REGION Network 2: DESCRIPTION
   // The block is used as a calling interface for the function blocks  
   // *   _Shiftmodel
   // *   _ProdDataCycleTimer
   // *   _ProdDataCounter
   // *   _ProdDataLimitValues
   // *   _ProdDataShiftCounter
   // or
   // *   _ProdDataShiftCounterOee, ShiftProductionTimes
   // 
   // **Calling interface**  
   // The block must be called once only in the cyclic program.  
   // 
   // The block is used as a calling interface for the function blocks  
   // *   _Shiftmodel
   // *   _ProdDataCycleTimer
   // *   _ProdDataCounter
   // *   _ProdDataLimitValues
   // *   _ProdDataShiftCounter
   // or
   // *   _ProdDataShiftCounterOee, ShiftProductionTimes
   // 
   // #### Additional information
   // 
   // #### Update info
   // 
   // #### Further documentations
   // 
   // ![Icon](_Icon/reference.PNG) 
   // 
   // See:  
   // ..\Library Types\LSicar_Shiftmodel.pdf  
   // ..\Library Types\LSicar_ProdDataCycleTimer.pdf  
   // ..\Library Types\LSicar_ProdDataCounter.pdf  
   // ..\Library Types\LSicar_ProdDataLimitValues.pdf  
   // ..\Library Types\LSicar_ProdDataShiftCounter.pdf  
   // ..\Library Types\LSicar_ProdDataShiftCounterOee.pdf  
   // ..\Library Types\LSicar_ShiftProductionTimes.pdf
END_REGION

REGION Network 3
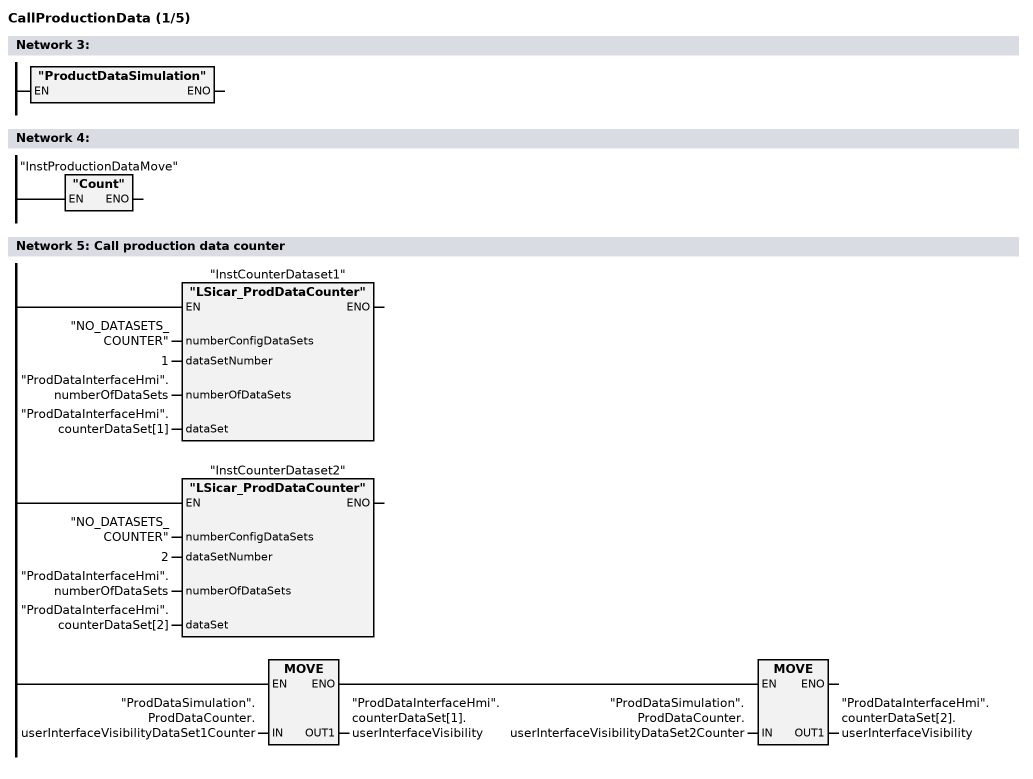
   RUNG wire#powerrail
      "ProductDataSimulation"()
   END_RUNG
   // the same network as SCL:
   "ProductDataSimulation"();
END_REGION

REGION Network 4
   RUNG wire#powerrail
      "InstProductionDataMove"()
   END_RUNG
   // the same network as SCL:
   "InstProductionDataMove"();   // "Count"
END_REGION

REGION Network 5: Call production data counter
   RUNG wire#powerrail
      "InstCounterDataset1"(numberConfigDataSets := "NO_DATASETS_COUNTER", dataSetNumber := 1, numberOfDataSets := "ProdDataInterfaceHmi".numberOfDataSets, dataSet := "ProdDataInterfaceHmi".counterDataSet[1])
   END_RUNG
   RUNG wire#powerrail
      "InstCounterDataset2"(numberConfigDataSets := "NO_DATASETS_COUNTER", dataSetNumber := 2, numberOfDataSets := "ProdDataInterfaceHmi".numberOfDataSets, dataSet := "ProdDataInterfaceHmi".counterDataSet[2])
   END_RUNG
   RUNG wire#powerrail
      Move(in := "ProdDataSimulation".ProdDataCounter.userInterfaceVisibilityDataSet1Counter, out1 => "ProdDataInterfaceHmi".counterDataSet[1].userInterfaceVisibility)
      Move(in := "ProdDataSimulation".ProdDataCounter.userInterfaceVisibilityDataSet2Counter, out1 => "ProdDataInterfaceHmi".counterDataSet[2].userInterfaceVisibility)
   END_RUNG
   // the same network as SCL:
   "InstCounterDataset1"(numberConfigDataSets := "NO_DATASETS_COUNTER",   // "LSicar_ProdDataCounter"
                         dataSetNumber := 1,
                         numberOfDataSets := "ProdDataInterfaceHmi".numberOfDataSets,
                         dataSet := "ProdDataInterfaceHmi".counterDataSet[1]);
   "InstCounterDataset2"(numberConfigDataSets := "NO_DATASETS_COUNTER",   // "LSicar_ProdDataCounter"
                         dataSetNumber := 2,
                         numberOfDataSets := "ProdDataInterfaceHmi".numberOfDataSets,
                         dataSet := "ProdDataInterfaceHmi".counterDataSet[2]);
   "ProdDataInterfaceHmi".counterDataSet[1].userInterfaceVisibility := "ProdDataSimulation".ProdDataCounter.userInterfaceVisibilityDataSet1Counter;
   "ProdDataInterfaceHmi".counterDataSet[2].userInterfaceVisibility := "ProdDataSimulation".ProdDataCounter.userInterfaceVisibilityDataSet2Counter;
END_REGION

REGION Network 6: Call production data cycle timer
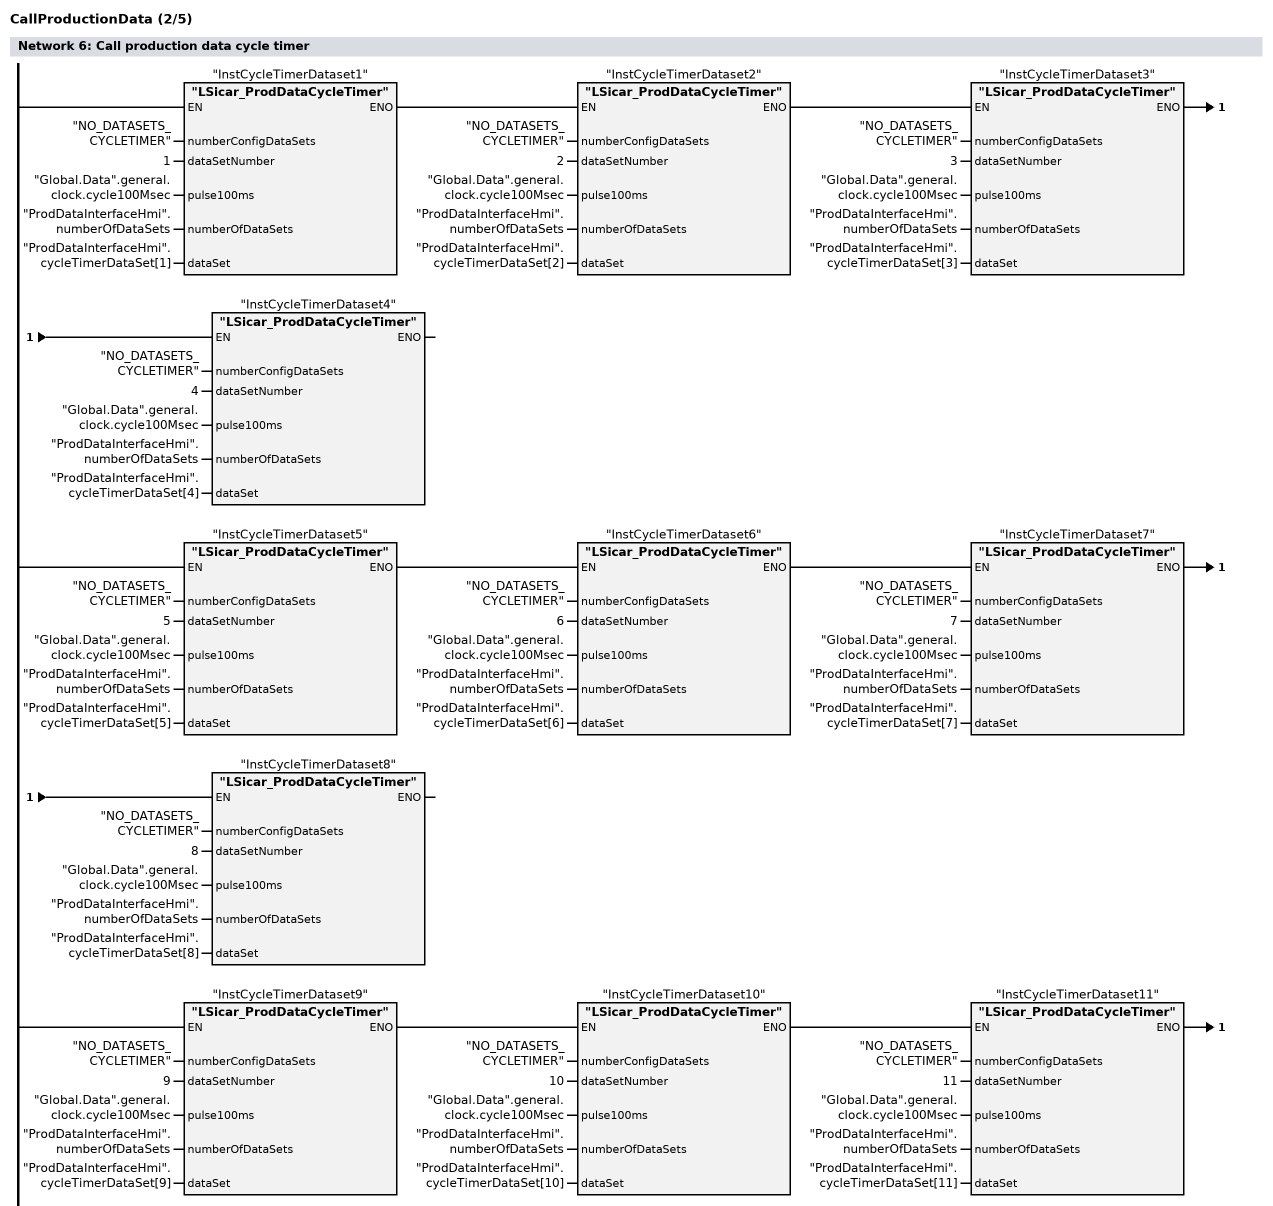
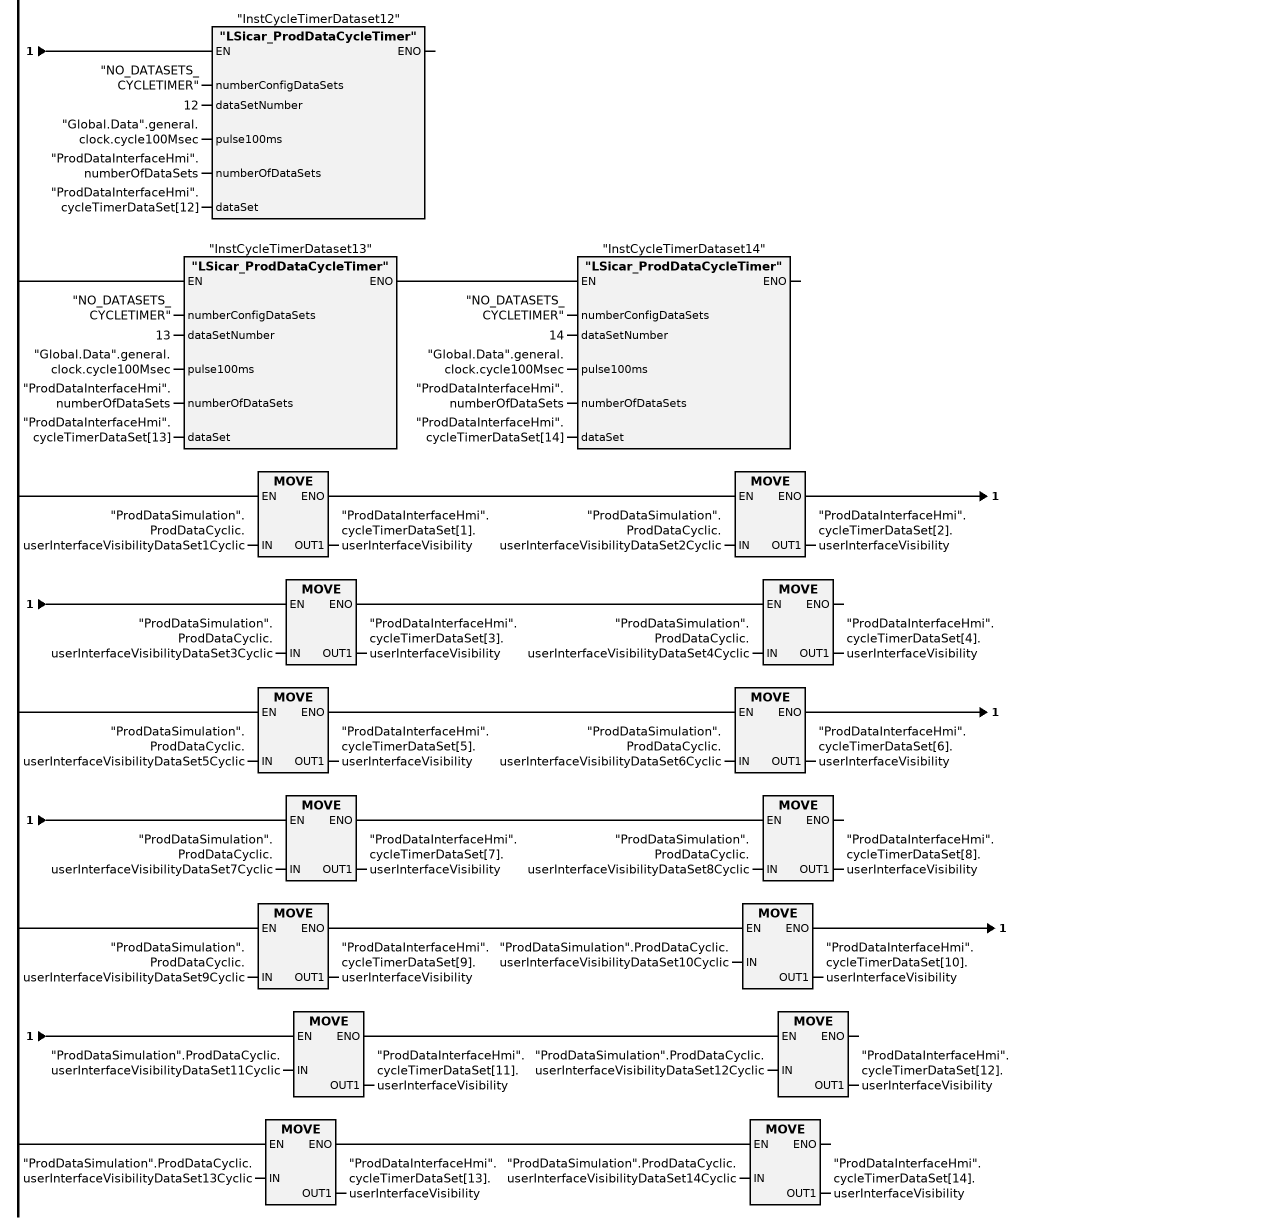
   RUNG wire#powerrail
      "InstCycleTimerDataset1"(numberConfigDataSets := "NO_DATASETS_CYCLETIMER", dataSetNumber := 1, pulse100ms := "Global.Data".general.clock.cycle100Msec, numberOfDataSets := "ProdDataInterfaceHmi".numberOfDataSets, dataSet := "ProdDataInterfaceHmi".cycleTimerDataSet[1])
      "InstCycleTimerDataset2"(numberConfigDataSets := "NO_DATASETS_CYCLETIMER", dataSetNumber := 2, pulse100ms := "Global.Data".general.clock.cycle100Msec, numberOfDataSets := "ProdDataInterfaceHmi".numberOfDataSets, dataSet := "ProdDataInterfaceHmi".cycleTimerDataSet[2])
      "InstCycleTimerDataset3"(numberConfigDataSets := "NO_DATASETS_CYCLETIMER", dataSetNumber := 3, pulse100ms := "Global.Data".general.clock.cycle100Msec, numberOfDataSets := "ProdDataInterfaceHmi".numberOfDataSets, dataSet := "ProdDataInterfaceHmi".cycleTimerDataSet[3])
      "InstCycleTimerDataset4"(numberConfigDataSets := "NO_DATASETS_CYCLETIMER", dataSetNumber := 4, pulse100ms := "Global.Data".general.clock.cycle100Msec, numberOfDataSets := "ProdDataInterfaceHmi".numberOfDataSets, dataSet := "ProdDataInterfaceHmi".cycleTimerDataSet[4])
   END_RUNG
   RUNG wire#powerrail
      "InstCycleTimerDataset5"(numberConfigDataSets := "NO_DATASETS_CYCLETIMER", dataSetNumber := 5, pulse100ms := "Global.Data".general.clock.cycle100Msec, numberOfDataSets := "ProdDataInterfaceHmi".numberOfDataSets, dataSet := "ProdDataInterfaceHmi".cycleTimerDataSet[5])
      "InstCycleTimerDataset6"(numberConfigDataSets := "NO_DATASETS_CYCLETIMER", dataSetNumber := 6, pulse100ms := "Global.Data".general.clock.cycle100Msec, numberOfDataSets := "ProdDataInterfaceHmi".numberOfDataSets, dataSet := "ProdDataInterfaceHmi".cycleTimerDataSet[6])
      "InstCycleTimerDataset7"(numberConfigDataSets := "NO_DATASETS_CYCLETIMER", dataSetNumber := 7, pulse100ms := "Global.Data".general.clock.cycle100Msec, numberOfDataSets := "ProdDataInterfaceHmi".numberOfDataSets, dataSet := "ProdDataInterfaceHmi".cycleTimerDataSet[7])
      "InstCycleTimerDataset8"(numberConfigDataSets := "NO_DATASETS_CYCLETIMER", dataSetNumber := 8, pulse100ms := "Global.Data".general.clock.cycle100Msec, numberOfDataSets := "ProdDataInterfaceHmi".numberOfDataSets, dataSet := "ProdDataInterfaceHmi".cycleTimerDataSet[8])
   END_RUNG
   RUNG wire#powerrail
      "InstCycleTimerDataset9"(numberConfigDataSets := "NO_DATASETS_CYCLETIMER", dataSetNumber := 9, pulse100ms := "Global.Data".general.clock.cycle100Msec, numberOfDataSets := "ProdDataInterfaceHmi".numberOfDataSets, dataSet := "ProdDataInterfaceHmi".cycleTimerDataSet[9])
      "InstCycleTimerDataset10"(numberConfigDataSets := "NO_DATASETS_CYCLETIMER", dataSetNumber := 10, pulse100ms := "Global.Data".general.clock.cycle100Msec, numberOfDataSets := "ProdDataInterfaceHmi".numberOfDataSets, dataSet := "ProdDataInterfaceHmi".cycleTimerDataSet[10])
      "InstCycleTimerDataset11"(numberConfigDataSets := "NO_DATASETS_CYCLETIMER", dataSetNumber := 11, pulse100ms := "Global.Data".general.clock.cycle100Msec, numberOfDataSets := "ProdDataInterfaceHmi".numberOfDataSets, dataSet := "ProdDataInterfaceHmi".cycleTimerDataSet[11])
      "InstCycleTimerDataset12"(numberConfigDataSets := "NO_DATASETS_CYCLETIMER", dataSetNumber := 12, pulse100ms := "Global.Data".general.clock.cycle100Msec, numberOfDataSets := "ProdDataInterfaceHmi".numberOfDataSets, dataSet := "ProdDataInterfaceHmi".cycleTimerDataSet[12])
   END_RUNG
   RUNG wire#powerrail
      "InstCycleTimerDataset13"(numberConfigDataSets := "NO_DATASETS_CYCLETIMER", dataSetNumber := 13, pulse100ms := "Global.Data".general.clock.cycle100Msec, numberOfDataSets := "ProdDataInterfaceHmi".numberOfDataSets, dataSet := "ProdDataInterfaceHmi".cycleTimerDataSet[13])
      "InstCycleTimerDataset14"(numberConfigDataSets := "NO_DATASETS_CYCLETIMER", dataSetNumber := 14, pulse100ms := "Global.Data".general.clock.cycle100Msec, numberOfDataSets := "ProdDataInterfaceHmi".numberOfDataSets, dataSet := "ProdDataInterfaceHmi".cycleTimerDataSet[14])
   END_RUNG
   RUNG wire#powerrail
      Move(in := "ProdDataSimulation".ProdDataCyclic.userInterfaceVisibilityDataSet1Cyclic, out1 => "ProdDataInterfaceHmi".cycleTimerDataSet[1].userInterfaceVisibility)
      Move(in := "ProdDataSimulation".ProdDataCyclic.userInterfaceVisibilityDataSet2Cyclic, out1 => "ProdDataInterfaceHmi".cycleTimerDataSet[2].userInterfaceVisibility)
      Move(in := "ProdDataSimulation".ProdDataCyclic.userInterfaceVisibilityDataSet3Cyclic, out1 => "ProdDataInterfaceHmi".cycleTimerDataSet[3].userInterfaceVisibility)
      Move(in := "ProdDataSimulation".ProdDataCyclic.userInterfaceVisibilityDataSet4Cyclic, out1 => "ProdDataInterfaceHmi".cycleTimerDataSet[4].userInterfaceVisibility)
   END_RUNG
   RUNG wire#powerrail
      Move(in := "ProdDataSimulation".ProdDataCyclic.userInterfaceVisibilityDataSet5Cyclic, out1 => "ProdDataInterfaceHmi".cycleTimerDataSet[5].userInterfaceVisibility)
      Move(in := "ProdDataSimulation".ProdDataCyclic.userInterfaceVisibilityDataSet6Cyclic, out1 => "ProdDataInterfaceHmi".cycleTimerDataSet[6].userInterfaceVisibility)
      Move(in := "ProdDataSimulation".ProdDataCyclic.userInterfaceVisibilityDataSet7Cyclic, out1 => "ProdDataInterfaceHmi".cycleTimerDataSet[7].userInterfaceVisibility)
      Move(in := "ProdDataSimulation".ProdDataCyclic.userInterfaceVisibilityDataSet8Cyclic, out1 => "ProdDataInterfaceHmi".cycleTimerDataSet[8].userInterfaceVisibility)
   END_RUNG
   RUNG wire#powerrail
      Move(in := "ProdDataSimulation".ProdDataCyclic.userInterfaceVisibilityDataSet9Cyclic, out1 => "ProdDataInterfaceHmi".cycleTimerDataSet[9].userInterfaceVisibility)
      Move(in := "ProdDataSimulation".ProdDataCyclic.userInterfaceVisibilityDataSet10Cyclic, out1 => "ProdDataInterfaceHmi".cycleTimerDataSet[10].userInterfaceVisibility)
      Move(in := "ProdDataSimulation".ProdDataCyclic.userInterfaceVisibilityDataSet11Cyclic, out1 => "ProdDataInterfaceHmi".cycleTimerDataSet[11].userInterfaceVisibility)
      Move(in := "ProdDataSimulation".ProdDataCyclic.userInterfaceVisibilityDataSet12Cyclic, out1 => "ProdDataInterfaceHmi".cycleTimerDataSet[12].userInterfaceVisibility)
   END_RUNG
   RUNG wire#powerrail
      Move(in := "ProdDataSimulation".ProdDataCyclic.userInterfaceVisibilityDataSet13Cyclic, out1 => "ProdDataInterfaceHmi".cycleTimerDataSet[13].userInterfaceVisibility)
      Move(in := "ProdDataSimulation".ProdDataCyclic.userInterfaceVisibilityDataSet14Cyclic, out1 => "ProdDataInterfaceHmi".cycleTimerDataSet[14].userInterfaceVisibility)
   END_RUNG
   // the same network as SCL:
   "InstCycleTimerDataset1"(numberConfigDataSets := "NO_DATASETS_CYCLETIMER",   // "LSicar_ProdDataCycleTimer"
                           dataSetNumber := 1,
                           pulse100ms := "Global.Data".general.clock.cycle100Msec,
                           numberOfDataSets := "ProdDataInterfaceHmi".numberOfDataSets,
                           dataSet := "ProdDataInterfaceHmi".cycleTimerDataSet[1],
                           ENO => #_w1);
   "InstCycleTimerDataset2"(EN := #_w1,   // "LSicar_ProdDataCycleTimer"
                           numberConfigDataSets := "NO_DATASETS_CYCLETIMER",
                           dataSetNumber := 2,
                           pulse100ms := "Global.Data".general.clock.cycle100Msec,
                           numberOfDataSets := "ProdDataInterfaceHmi".numberOfDataSets,
                           dataSet := "ProdDataInterfaceHmi".cycleTimerDataSet[2],
                           ENO => #_w2);
   "InstCycleTimerDataset3"(EN := #_w2,   // "LSicar_ProdDataCycleTimer"
                           numberConfigDataSets := "NO_DATASETS_CYCLETIMER",
                           dataSetNumber := 3,
                           pulse100ms := "Global.Data".general.clock.cycle100Msec,
                           numberOfDataSets := "ProdDataInterfaceHmi".numberOfDataSets,
                           dataSet := "ProdDataInterfaceHmi".cycleTimerDataSet[3],
                           ENO => #_w3);
   IF #_w3 THEN
       "InstCycleTimerDataset4"(numberConfigDataSets := "NO_DATASETS_CYCLETIMER",   // "LSicar_ProdDataCycleTimer"
                               dataSetNumber := 4,
                               pulse100ms := "Global.Data".general.clock.cycle100Msec,
                               numberOfDataSets := "ProdDataInterfaceHmi".numberOfDataSets,
                               dataSet := "ProdDataInterfaceHmi".cycleTimerDataSet[4]);
   END_IF;
   "InstCycleTimerDataset5"(numberConfigDataSets := "NO_DATASETS_CYCLETIMER",   // "LSicar_ProdDataCycleTimer"
                           dataSetNumber := 5,
                           pulse100ms := "Global.Data".general.clock.cycle100Msec,
                           numberOfDataSets := "ProdDataInterfaceHmi".numberOfDataSets,
                           dataSet := "ProdDataInterfaceHmi".cycleTimerDataSet[5],
                           ENO => #_w4);
   "InstCycleTimerDataset6"(EN := #_w4,   // "LSicar_ProdDataCycleTimer"
                           numberConfigDataSets := "NO_DATASETS_CYCLETIMER",
                           dataSetNumber := 6,
                           pulse100ms := "Global.Data".general.clock.cycle100Msec,
                           numberOfDataSets := "ProdDataInterfaceHmi".numberOfDataSets,
                           dataSet := "ProdDataInterfaceHmi".cycleTimerDataSet[6],
                           ENO => #_w5);
   "InstCycleTimerDataset7"(EN := #_w5,   // "LSicar_ProdDataCycleTimer"
                           numberConfigDataSets := "NO_DATASETS_CYCLETIMER",
                           dataSetNumber := 7,
                           pulse100ms := "Global.Data".general.clock.cycle100Msec,
                           numberOfDataSets := "ProdDataInterfaceHmi".numberOfDataSets,
                           dataSet := "ProdDataInterfaceHmi".cycleTimerDataSet[7],
                           ENO => #_w6);
   IF #_w6 THEN
       "InstCycleTimerDataset8"(numberConfigDataSets := "NO_DATASETS_CYCLETIMER",   // "LSicar_ProdDataCycleTimer"
                               dataSetNumber := 8,
                               pulse100ms := "Global.Data".general.clock.cycle100Msec,
                               numberOfDataSets := "ProdDataInterfaceHmi".numberOfDataSets,
                               dataSet := "ProdDataInterfaceHmi".cycleTimerDataSet[8]);
   END_IF;
   "InstCycleTimerDataset9"(numberConfigDataSets := "NO_DATASETS_CYCLETIMER",   // "LSicar_ProdDataCycleTimer"
                           dataSetNumber := 9,
                           pulse100ms := "Global.Data".general.clock.cycle100Msec,
                           numberOfDataSets := "ProdDataInterfaceHmi".numberOfDataSets,
                           dataSet := "ProdDataInterfaceHmi".cycleTimerDataSet[9],
                           ENO => #_w7);
   "InstCycleTimerDataset10"(EN := #_w7,   // "LSicar_ProdDataCycleTimer"
                           numberConfigDataSets := "NO_DATASETS_CYCLETIMER",
                           dataSetNumber := 10,
                           pulse100ms := "Global.Data".general.clock.cycle100Msec,
                           numberOfDataSets := "ProdDataInterfaceHmi".numberOfDataSets,
                           dataSet := "ProdDataInterfaceHmi".cycleTimerDataSet[10],
                           ENO => #_w8);
   "InstCycleTimerDataset11"(EN := #_w8,   // "LSicar_ProdDataCycleTimer"
                           numberConfigDataSets := "NO_DATASETS_CYCLETIMER",
                           dataSetNumber := 11,
                           pulse100ms := "Global.Data".general.clock.cycle100Msec,
                           numberOfDataSets := "ProdDataInterfaceHmi".numberOfDataSets,
                           dataSet := "ProdDataInterfaceHmi".cycleTimerDataSet[11],
                           ENO => #_w9);
   IF #_w9 THEN
       "InstCycleTimerDataset12"(numberConfigDataSets := "NO_DATASETS_CYCLETIMER",   // "LSicar_ProdDataCycleTimer"
                               dataSetNumber := 12,
                               pulse100ms := "Global.Data".general.clock.cycle100Msec,
                               numberOfDataSets := "ProdDataInterfaceHmi".numberOfDataSets,
                               dataSet := "ProdDataInterfaceHmi".cycleTimerDataSet[12]);
   END_IF;
   "InstCycleTimerDataset13"(numberConfigDataSets := "NO_DATASETS_CYCLETIMER",   // "LSicar_ProdDataCycleTimer"
                           dataSetNumber := 13,
                           pulse100ms := "Global.Data".general.clock.cycle100Msec,
                           numberOfDataSets := "ProdDataInterfaceHmi".numberOfDataSets,
                           dataSet := "ProdDataInterfaceHmi".cycleTimerDataSet[13],
                           ENO => #_w10);
   IF #_w10 THEN
       "InstCycleTimerDataset14"(numberConfigDataSets := "NO_DATASETS_CYCLETIMER",   // "LSicar_ProdDataCycleTimer"
                               dataSetNumber := 14,
                               pulse100ms := "Global.Data".general.clock.cycle100Msec,
                               numberOfDataSets := "ProdDataInterfaceHmi".numberOfDataSets,
                               dataSet := "ProdDataInterfaceHmi".cycleTimerDataSet[14]);
   END_IF;
   "ProdDataInterfaceHmi".cycleTimerDataSet[1].userInterfaceVisibility := "ProdDataSimulation".ProdDataCyclic.userInterfaceVisibilityDataSet1Cyclic;
   "ProdDataInterfaceHmi".cycleTimerDataSet[2].userInterfaceVisibility := "ProdDataSimulation".ProdDataCyclic.userInterfaceVisibilityDataSet2Cyclic;
   "ProdDataInterfaceHmi".cycleTimerDataSet[3].userInterfaceVisibility := "ProdDataSimulation".ProdDataCyclic.userInterfaceVisibilityDataSet3Cyclic;
   "ProdDataInterfaceHmi".cycleTimerDataSet[4].userInterfaceVisibility := "ProdDataSimulation".ProdDataCyclic.userInterfaceVisibilityDataSet4Cyclic;
   "ProdDataInterfaceHmi".cycleTimerDataSet[5].userInterfaceVisibility := "ProdDataSimulation".ProdDataCyclic.userInterfaceVisibilityDataSet5Cyclic;
   "ProdDataInterfaceHmi".cycleTimerDataSet[6].userInterfaceVisibility := "ProdDataSimulation".ProdDataCyclic.userInterfaceVisibilityDataSet6Cyclic;
   "ProdDataInterfaceHmi".cycleTimerDataSet[7].userInterfaceVisibility := "ProdDataSimulation".ProdDataCyclic.userInterfaceVisibilityDataSet7Cyclic;
   "ProdDataInterfaceHmi".cycleTimerDataSet[8].userInterfaceVisibility := "ProdDataSimulation".ProdDataCyclic.userInterfaceVisibilityDataSet8Cyclic;
   "ProdDataInterfaceHmi".cycleTimerDataSet[9].userInterfaceVisibility := "ProdDataSimulation".ProdDataCyclic.userInterfaceVisibilityDataSet9Cyclic;
   "ProdDataInterfaceHmi".cycleTimerDataSet[10].userInterfaceVisibility := "ProdDataSimulation".ProdDataCyclic.userInterfaceVisibilityDataSet10Cyclic;
   "ProdDataInterfaceHmi".cycleTimerDataSet[11].userInterfaceVisibility := "ProdDataSimulation".ProdDataCyclic.userInterfaceVisibilityDataSet11Cyclic;
   "ProdDataInterfaceHmi".cycleTimerDataSet[12].userInterfaceVisibility := "ProdDataSimulation".ProdDataCyclic.userInterfaceVisibilityDataSet12Cyclic;
   "ProdDataInterfaceHmi".cycleTimerDataSet[13].userInterfaceVisibility := "ProdDataSimulation".ProdDataCyclic.userInterfaceVisibilityDataSet13Cyclic;
   "ProdDataInterfaceHmi".cycleTimerDataSet[14].userInterfaceVisibility := "ProdDataSimulation".ProdDataCyclic.userInterfaceVisibilityDataSet14Cyclic;
END_REGION

REGION Network 7: Call production data limit values
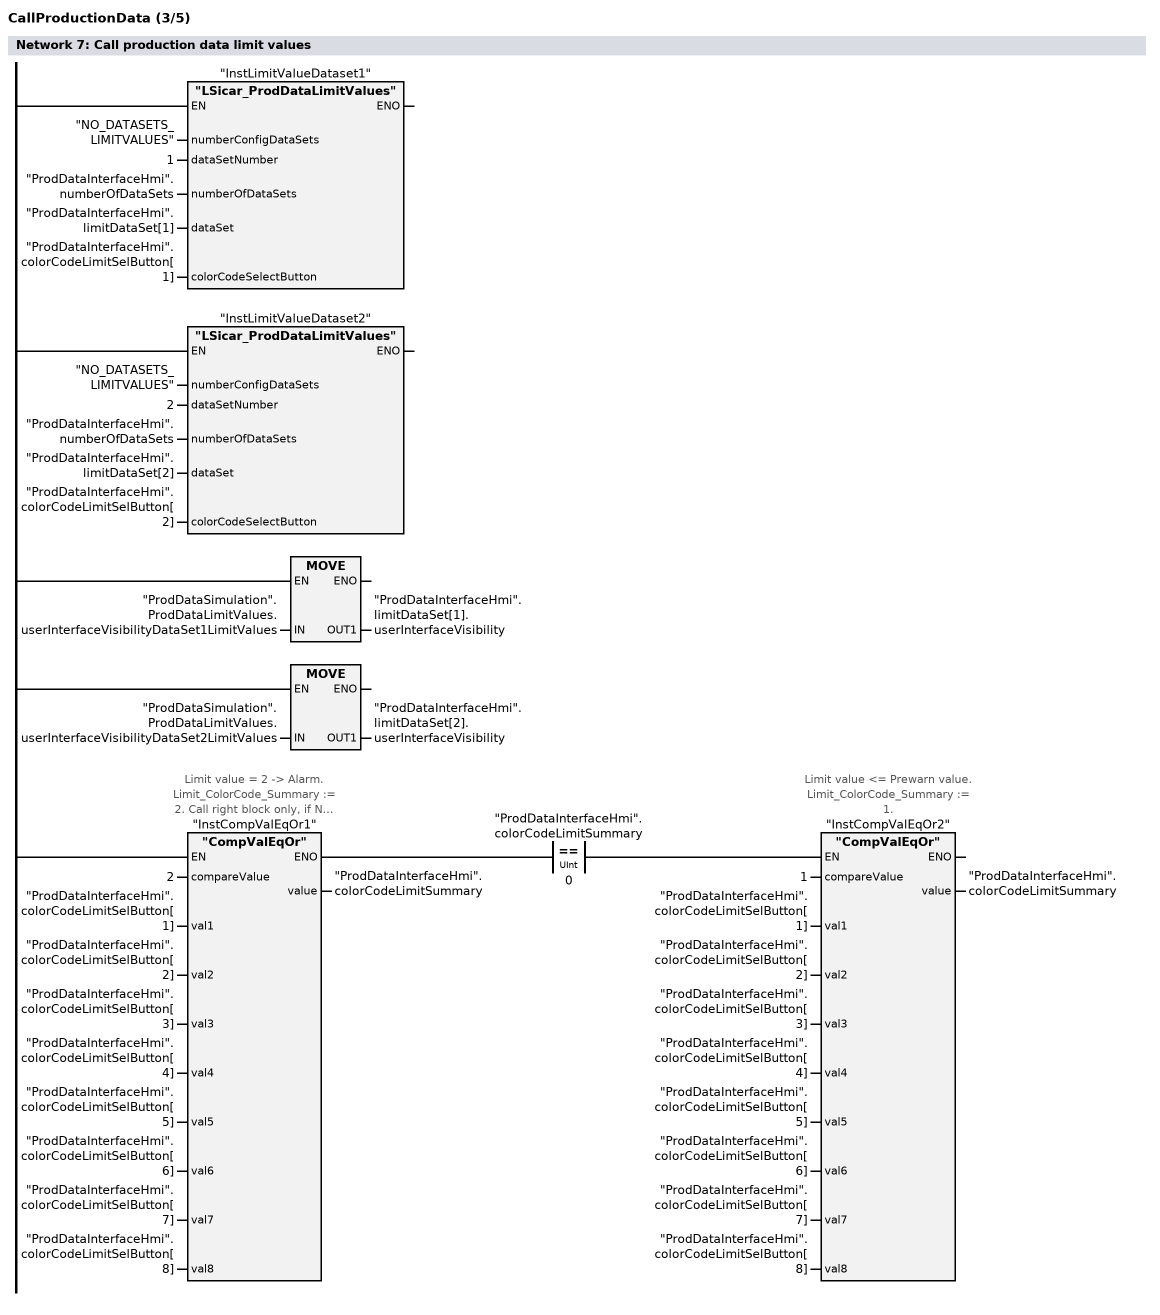
   RUNG wire#powerrail
      "InstLimitValueDataset1"(numberConfigDataSets := "NO_DATASETS_LIMITVALUES", dataSetNumber := 1, numberOfDataSets := "ProdDataInterfaceHmi".numberOfDataSets, dataSet := "ProdDataInterfaceHmi".limitDataSet[1], colorCodeSelectButton := "ProdDataInterfaceHmi".colorCodeLimitSelButton[1])
   END_RUNG
   RUNG wire#powerrail
      "InstLimitValueDataset2"(numberConfigDataSets := "NO_DATASETS_LIMITVALUES", dataSetNumber := 2, numberOfDataSets := "ProdDataInterfaceHmi".numberOfDataSets, dataSet := "ProdDataInterfaceHmi".limitDataSet[2], colorCodeSelectButton := "ProdDataInterfaceHmi".colorCodeLimitSelButton[2])
   END_RUNG
   RUNG wire#powerrail
      Move(in := "ProdDataSimulation".ProdDataLimitValues.userInterfaceVisibilityDataSet1LimitValues, out1 => "ProdDataInterfaceHmi".limitDataSet[1].userInterfaceVisibility)
   END_RUNG
   RUNG wire#powerrail
      Move(in := "ProdDataSimulation".ProdDataLimitValues.userInterfaceVisibilityDataSet2LimitValues, out1 => "ProdDataInterfaceHmi".limitDataSet[2].userInterfaceVisibility)
   END_RUNG
   RUNG wire#powerrail
      "InstCompValEqOr1"(compareValue := 2, val1 := "ProdDataInterfaceHmi".colorCodeLimitSelButton[1], val2 := "ProdDataInterfaceHmi".colorCodeLimitSelButton[2], val3 := "ProdDataInterfaceHmi".colorCodeLimitSelButton[3], val4 := "ProdDataInterfaceHmi".colorCodeLimitSelButton[4], val5 := "ProdDataInterfaceHmi".colorCodeLimitSelButton[5], val6 := "ProdDataInterfaceHmi".colorCodeLimitSelButton[6], val7 := "ProdDataInterfaceHmi".colorCodeLimitSelButton[7], val8 := "ProdDataInterfaceHmi".colorCodeLimitSelButton[8], value => "ProdDataInterfaceHmi".colorCodeLimitSummary)   // Limit value = 2 -> Alarm. Limit_ColorCode_Summary := 2. Call right block only, if NO alarm (VALUE = 0) is pending here; alarm is higher prior.
      { S7_Templates := "SrcType := UInt" } EQ_Contact(in1 := "ProdDataInterfaceHmi".colorCodeLimitSummary, in2 := 0)
      "InstCompValEqOr2"(compareValue := 1, val1 := "ProdDataInterfaceHmi".colorCodeLimitSelButton[1], val2 := "ProdDataInterfaceHmi".colorCodeLimitSelButton[2], val3 := "ProdDataInterfaceHmi".colorCodeLimitSelButton[3], val4 := "ProdDataInterfaceHmi".colorCodeLimitSelButton[4], val5 := "ProdDataInterfaceHmi".colorCodeLimitSelButton[5], val6 := "ProdDataInterfaceHmi".colorCodeLimitSelButton[6], val7 := "ProdDataInterfaceHmi".colorCodeLimitSelButton[7], val8 := "ProdDataInterfaceHmi".colorCodeLimitSelButton[8], value => "ProdDataInterfaceHmi".colorCodeLimitSummary)   // Limit value <= Prewarn value. Limit_ColorCode_Summary := 1.
   END_RUNG
   // the same network as SCL:
   "InstLimitValueDataset1"(numberConfigDataSets := "NO_DATASETS_LIMITVALUES",   // "LSicar_ProdDataLimitValues"
                           dataSetNumber := 1,
                           numberOfDataSets := "ProdDataInterfaceHmi".numberOfDataSets,
                           dataSet := "ProdDataInterfaceHmi".limitDataSet[1],
                           colorCodeSelectButton := "ProdDataInterfaceHmi".colorCodeLimitSelButton[1]);
   "InstLimitValueDataset2"(numberConfigDataSets := "NO_DATASETS_LIMITVALUES",   // "LSicar_ProdDataLimitValues"
                           dataSetNumber := 2,
                           numberOfDataSets := "ProdDataInterfaceHmi".numberOfDataSets,
                           dataSet := "ProdDataInterfaceHmi".limitDataSet[2],
                           colorCodeSelectButton := "ProdDataInterfaceHmi".colorCodeLimitSelButton[2]);
   "ProdDataInterfaceHmi".limitDataSet[1].userInterfaceVisibility := "ProdDataSimulation".ProdDataLimitValues.userInterfaceVisibilityDataSet1LimitValues;
   "ProdDataInterfaceHmi".limitDataSet[2].userInterfaceVisibility := "ProdDataSimulation".ProdDataLimitValues.userInterfaceVisibilityDataSet2LimitValues;
   "InstCompValEqOr1"(compareValue := 2,   // "CompValEqOr": Limit value = 2 -> Alarm. Limit_ColorCode_Summary := 2. Call right block only, if NO alarm (VALUE = 0) is pending here; alarm is higher prior.
                      val1 := "ProdDataInterfaceHmi".colorCodeLimitSelButton[1],
                      val2 := "ProdDataInterfaceHmi".colorCodeLimitSelButton[2],
                      val3 := "ProdDataInterfaceHmi".colorCodeLimitSelButton[3],
                      val4 := "ProdDataInterfaceHmi".colorCodeLimitSelButton[4],
                      val5 := "ProdDataInterfaceHmi".colorCodeLimitSelButton[5],
                      val6 := "ProdDataInterfaceHmi".colorCodeLimitSelButton[6],
                      val7 := "ProdDataInterfaceHmi".colorCodeLimitSelButton[7],
                      val8 := "ProdDataInterfaceHmi".colorCodeLimitSelButton[8],
                      value => "ProdDataInterfaceHmi".colorCodeLimitSummary,
                      ENO => #_w1);
   IF #_w1 AND ("ProdDataInterfaceHmi".colorCodeLimitSummary = 0) THEN
       "InstCompValEqOr2"(compareValue := 1,   // "CompValEqOr": Limit value <= Prewarn value. Limit_ColorCode_Summary := 1.
                          val1 := "ProdDataInterfaceHmi".colorCodeLimitSelButton[1],
                          val2 := "ProdDataInterfaceHmi".colorCodeLimitSelButton[2],
                          val3 := "ProdDataInterfaceHmi".colorCodeLimitSelButton[3],
                          val4 := "ProdDataInterfaceHmi".colorCodeLimitSelButton[4],
                          val5 := "ProdDataInterfaceHmi".colorCodeLimitSelButton[5],
                          val6 := "ProdDataInterfaceHmi".colorCodeLimitSelButton[6],
                          val7 := "ProdDataInterfaceHmi".colorCodeLimitSelButton[7],
                          val8 := "ProdDataInterfaceHmi".colorCodeLimitSelButton[8],
                          value => "ProdDataInterfaceHmi".colorCodeLimitSummary);
   END_IF;
END_REGION

REGION Network 8: Call production data shift counter
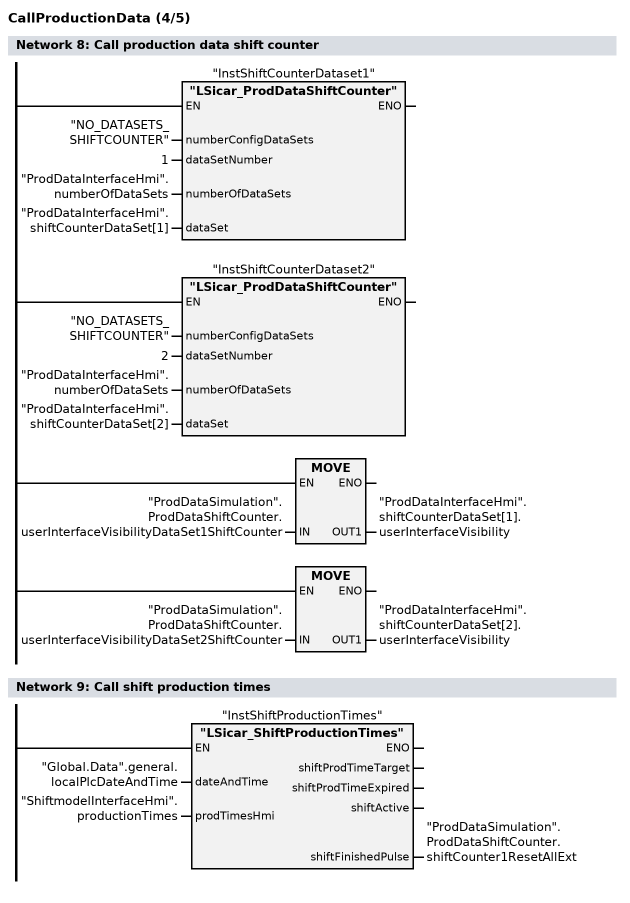
   RUNG wire#powerrail
      "InstShiftCounterDataset1"(numberConfigDataSets := "NO_DATASETS_SHIFTCOUNTER", dataSetNumber := 1, numberOfDataSets := "ProdDataInterfaceHmi".numberOfDataSets, dataSet := "ProdDataInterfaceHmi".shiftCounterDataSet[1])
   END_RUNG
   RUNG wire#powerrail
      "InstShiftCounterDataset2"(numberConfigDataSets := "NO_DATASETS_SHIFTCOUNTER", dataSetNumber := 2, numberOfDataSets := "ProdDataInterfaceHmi".numberOfDataSets, dataSet := "ProdDataInterfaceHmi".shiftCounterDataSet[2])
   END_RUNG
   RUNG wire#powerrail
      Move(in := "ProdDataSimulation".ProdDataShiftCounter.userInterfaceVisibilityDataSet1ShiftCounter, out1 => "ProdDataInterfaceHmi".shiftCounterDataSet[1].userInterfaceVisibility)
   END_RUNG
   RUNG wire#powerrail
      Move(in := "ProdDataSimulation".ProdDataShiftCounter.userInterfaceVisibilityDataSet2ShiftCounter, out1 => "ProdDataInterfaceHmi".shiftCounterDataSet[2].userInterfaceVisibility)
   END_RUNG
   // the same network as SCL:
   "InstShiftCounterDataset1"(numberConfigDataSets := "NO_DATASETS_SHIFTCOUNTER",   // "LSicar_ProdDataShiftCounter"
                           dataSetNumber := 1,
                           numberOfDataSets := "ProdDataInterfaceHmi".numberOfDataSets,
                           dataSet := "ProdDataInterfaceHmi".shiftCounterDataSet[1]);
   "InstShiftCounterDataset2"(numberConfigDataSets := "NO_DATASETS_SHIFTCOUNTER",   // "LSicar_ProdDataShiftCounter"
                           dataSetNumber := 2,
                           numberOfDataSets := "ProdDataInterfaceHmi".numberOfDataSets,
                           dataSet := "ProdDataInterfaceHmi".shiftCounterDataSet[2]);
   "ProdDataInterfaceHmi".shiftCounterDataSet[1].userInterfaceVisibility := "ProdDataSimulation".ProdDataShiftCounter.userInterfaceVisibilityDataSet1ShiftCounter;
   "ProdDataInterfaceHmi".shiftCounterDataSet[2].userInterfaceVisibility := "ProdDataSimulation".ProdDataShiftCounter.userInterfaceVisibilityDataSet2ShiftCounter;
END_REGION

REGION Network 9: Call shift production times
   RUNG wire#powerrail
      "InstShiftProductionTimes"(dateAndTime := "Global.Data".general.localPlcDateAndTime, prodTimesHmi := "ShiftmodelInterfaceHmi".productionTimes, shiftProdTimeTarget =>, shiftProdTimeExpired =>, shiftActive =>, shiftFinishedPulse => "ProdDataSimulation".ProdDataShiftCounter.shiftCounter1ResetAllExt)
   END_RUNG
   // the same network as SCL:
   "InstShiftProductionTimes"(dateAndTime := "Global.Data".general.localPlcDateAndTime,   // "LSicar_ShiftProductionTimes"
                           prodTimesHmi := "ShiftmodelInterfaceHmi".productionTimes,
                           shiftFinishedPulse => "ProdDataSimulation".ProdDataShiftCounter.shiftCounter1ResetAllExt);
END_REGION

REGION Network 10: Call production data shift counter OEE
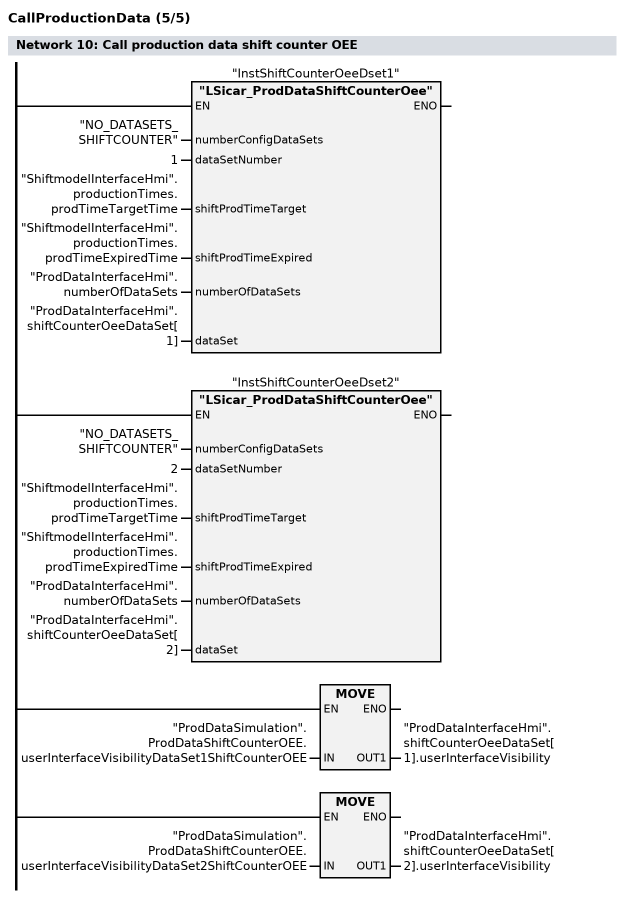
   RUNG wire#powerrail
      "InstShiftCounterOeeDset1"(numberConfigDataSets := "NO_DATASETS_SHIFTCOUNTER", dataSetNumber := 1, shiftProdTimeTarget := "ShiftmodelInterfaceHmi".productionTimes.prodTimeTargetTime, shiftProdTimeExpired := "ShiftmodelInterfaceHmi".productionTimes.prodTimeExpiredTime, numberOfDataSets := "ProdDataInterfaceHmi".numberOfDataSets, dataSet := "ProdDataInterfaceHmi".shiftCounterOeeDataSet[1])
   END_RUNG
   RUNG wire#powerrail
      "InstShiftCounterOeeDset2"(numberConfigDataSets := "NO_DATASETS_SHIFTCOUNTER", dataSetNumber := 2, shiftProdTimeTarget := "ShiftmodelInterfaceHmi".productionTimes.prodTimeTargetTime, shiftProdTimeExpired := "ShiftmodelInterfaceHmi".productionTimes.prodTimeExpiredTime, numberOfDataSets := "ProdDataInterfaceHmi".numberOfDataSets, dataSet := "ProdDataInterfaceHmi".shiftCounterOeeDataSet[2])
   END_RUNG
   RUNG wire#powerrail
      Move(in := "ProdDataSimulation".ProdDataShiftCounterOEE.userInterfaceVisibilityDataSet1ShiftCounterOEE, out1 => "ProdDataInterfaceHmi".shiftCounterOeeDataSet[1].userInterfaceVisibility)
   END_RUNG
   RUNG wire#powerrail
      Move(in := "ProdDataSimulation".ProdDataShiftCounterOEE.userInterfaceVisibilityDataSet2ShiftCounterOEE, out1 => "ProdDataInterfaceHmi".shiftCounterOeeDataSet[2].userInterfaceVisibility)
   END_RUNG
   // the same network as SCL:
   "InstShiftCounterOeeDset1"(numberConfigDataSets := "NO_DATASETS_SHIFTCOUNTER",   // "LSicar_ProdDataShiftCounterOee"
                           dataSetNumber := 1,
                           shiftProdTimeTarget := "ShiftmodelInterfaceHmi".productionTimes.prodTimeTargetTime,
                           shiftProdTimeExpired := "ShiftmodelInterfaceHmi".productionTimes.prodTimeExpiredTime,
                           numberOfDataSets := "ProdDataInterfaceHmi".numberOfDataSets,
                           dataSet := "ProdDataInterfaceHmi".shiftCounterOeeDataSet[1]);
   "InstShiftCounterOeeDset2"(numberConfigDataSets := "NO_DATASETS_SHIFTCOUNTER",   // "LSicar_ProdDataShiftCounterOee"
                           dataSetNumber := 2,
                           shiftProdTimeTarget := "ShiftmodelInterfaceHmi".productionTimes.prodTimeTargetTime,
                           shiftProdTimeExpired := "ShiftmodelInterfaceHmi".productionTimes.prodTimeExpiredTime,
                           numberOfDataSets := "ProdDataInterfaceHmi".numberOfDataSets,
                           dataSet := "ProdDataInterfaceHmi".shiftCounterOeeDataSet[2]);
   "ProdDataInterfaceHmi".shiftCounterOeeDataSet[1].userInterfaceVisibility := "ProdDataSimulation".ProdDataShiftCounterOEE.userInterfaceVisibilityDataSet1ShiftCounterOEE;
   "ProdDataInterfaceHmi".shiftCounterOeeDataSet[2].userInterfaceVisibility := "ProdDataSimulation".ProdDataShiftCounterOEE.userInterfaceVisibilityDataSet2ShiftCounterOEE;
END_REGION
END_FUNCTION

FUNCTION "ProductDataSimulation" : Void
{ S7_Optimized_Access := 'TRUE' ; Published := 'FALSE' }
VERSION : 0.1
//Block for simulate the Production Counter

BEGIN
	REGION BLOCK INFO HEADER
	    //===============================================================================
	    // Siemens AG / (c)Copyright 2023
	    //-------------------------------------------------------------------------------
	    // Title:            ProductDataSimulation (FC 4)
	    // Comment/Function: Block for simulate the Production Counter
	    // Library/Family:   Automation Framework
	    // Author:           -
	    // Tested with:      -
	    // Engineering:      TIA Portal V19
	    // Restrictions:     -
	    // Requirements:     -
	    //-------------------------------------------------------------------------------
	    // Change log table:
	    // Version  | Date       | Expert in charge              | Changes applied
	    //----------|------------|-------------------------------|-----------------------------
	    // 01.00.00 | 11.12.2023 |Siemens Industry Online Support| First released version
	    //===============================================================================    
	END_REGION
	
	REGION DESCRIPTION
	   (/*
	 This module is used to simulate the Production Counter:
	*  ProdDataCounter
	*  ProdDataCycleTimer
	*  ProdDataLimitValues
	*  ProdDataShiftCounter
	*  ProdDataShiftCounterOEE
	    
	The data in the data block ("ProdDataSimulation_ProdData") are written to the parameters in The "ProdDataInterfaceHmi".
	This allows the visual representation of the counters be displayed
	*/) 
	    
	    
	END_REGION
	REGION ProdDataCounter
	
	    // Implement an example counter for PrdDataCounter 1 and ProdDataCounter 2
	    IF "ProdDataSimulation".ProdDataCounter.ProdDataEnable THEN
	        
	        // ProdDataCounter 1
	        "ProdDataInterfaceHmi".counterDataSet[1].control[1].countUp := "ProdDataSimulation".ProdDataCounter.ProdDataCounter1Up1;
	        "ProdDataInterfaceHmi".counterDataSet[1].control[1].countDown := "ProdDataSimulation".ProdDataCounter.ProdDataCounter1Down1;
	        "ProdDataInterfaceHmi".counterDataSet[1].control[2].countUp := "ProdDataSimulation".ProdDataCounter.ProdDataCounter1Up2;
	        "ProdDataInterfaceHmi".counterDataSet[1].control[2].countDown := "ProdDataSimulation".ProdDataCounter.ProdDataCounter1Down2;
	        "ProdDataInterfaceHmi".counterDataSet[1].control[1].reset := "ProdDataSimulation".ProdDataCounter.ProdDataCounter1Reset1;
	        "ProdDataInterfaceHmi".counterDataSet[1].control[2].reset := "ProdDataSimulation".ProdDataCounter.ProdDataCounter1Reset2;
	        "ProdDataInterfaceHmi".counterDataSet[1].resetAllExt := "ProdDataSimulation".ProdDataCounter.ProdDataCounter1ResetAll;
	        
	        // ProdDataCounter 2
	        (* "ProdDataInterfaceHmi".counterDataSet[2].control[1].countUp := "ProdDataSimulation".ProdDataCounter.ProdDataCounter2Up1;
	        "ProdDataInterfaceHmi".counterDataSet[2].control[1].countDown := "ProdDataSimulation".ProdDataCounter.ProdDataCounter2Down1;
	        "ProdDataInterfaceHmi".counterDataSet[2].control[2].countUp := "ProdDataSimulation".ProdDataCounter.ProdDataCounter2Up2;
	        "ProdDataInterfaceHmi".counterDataSet[2].control[2].countDown := "ProdDataSimulation".ProdDataCounter.ProdDataCounter2Down2;
	        "ProdDataInterfaceHmi".counterDataSet[2].control[1].reset := "ProdDataSimulation".ProdDataCounter.ProdDataCounter2Reset1;
	        "ProdDataInterfaceHmi".counterDataSet[2].control[2].reset := "ProdDataSimulation".ProdDataCounter.ProdDataCounter2Reset2;
	        "ProdDataInterfaceHmi".counterDataSet[2].resetAllExt := "ProdDataSimulation".ProdDataCounter.ProdDataCounter2ResetAll; *)
	        
	        //Via the user interface „.userInterfaceVisibility“ [DWord] individual values can be hidden in the visualization
	        "ProdDataInterfaceHmi".counterDataSet[1].userInterfaceVisibility := "ProdDataSimulation".ProdDataCounter.userInterfaceVisibilityDataSet1Counter;
	        //"ProdDataInterfaceHmi".counterDataSet[2].userInterfaceVisibility := "ProdDataSimulation".ProdDataCounter.userInterfaceVisibilityDataSet2Counter;
	    END_IF;
	    
	END_REGION
	
	REGION CycleTimer
	    // Example to demonstrate and test the functionality of the cycle timer
	    IF "ProdDataSimulation".ProdDataCyclic.cyclicTimerEnable THEN
	        
	        "ProdDataInterfaceHmi".cycleTimerDataSet[1].control[1].run := "ProdDataSimulation".ProdDataCyclic.cycleTimer1Run1;
	        "ProdDataInterfaceHmi".cycleTimerDataSet[1].control[1].hold := "ProdDataSimulation".ProdDataCyclic.cycleTimer1Hold1;
	        "ProdDataInterfaceHmi".cycleTimerDataSet[1].control[1].reset := "ProdDataSimulation".ProdDataCyclic.cycleTimer1Reset1;
	        "ProdDataInterfaceHmi".cycleTimerDataSet[1].control[2].run := "ProdDataSimulation".ProdDataCyclic.cycleTimer1Run2;
	        "ProdDataInterfaceHmi".cycleTimerDataSet[1].control[2].hold := "ProdDataSimulation".ProdDataCyclic.cycleTimer1Hold2;
	        "ProdDataInterfaceHmi".cycleTimerDataSet[1].control[2].reset := "ProdDataSimulation".ProdDataCyclic.cycleTimer1Reset2;
	        "ProdDataInterfaceHmi".cycleTimerDataSet[2].control[1].run := "ProdDataSimulation".ProdDataCyclic.cycleTimer2Run1;
	        "ProdDataInterfaceHmi".cycleTimerDataSet[2].control[1].hold := "ProdDataSimulation".ProdDataCyclic.cycleTimer2Hold1;
	        "ProdDataInterfaceHmi".cycleTimerDataSet[2].control[1].reset := "ProdDataSimulation".ProdDataCyclic.cycleTimer2Reset1;
	        "ProdDataInterfaceHmi".cycleTimerDataSet[2].control[2].run := "ProdDataSimulation".ProdDataCyclic.cycleTimer2Run2;
	        "ProdDataInterfaceHmi".cycleTimerDataSet[2].control[2].hold := "ProdDataSimulation".ProdDataCyclic.cycleTimer2Hold2;
	        "ProdDataInterfaceHmi".cycleTimerDataSet[2].control[2].reset := "ProdDataSimulation".ProdDataCyclic.cycleTimer2Reset2;
	        "ProdDataInterfaceHmi".cycleTimerDataSet[1].resetAverageAllExt := "ProdDataSimulation".ProdDataCyclic.cycleTimer1ResetAll;
	        "ProdDataInterfaceHmi".cycleTimerDataSet[2].resetAverageAllExt := "ProdDataSimulation".ProdDataCyclic.cycleTimer2ResetAll;
	        
	        //Via the user interface „.userInterfaceVisibility“ [DWord] individual values can be hidden in the visualization
	        "ProdDataInterfaceHmi".cycleTimerDataSet[1].userInterfaceVisibility := "ProdDataSimulation".ProdDataCyclic.userInterfaceVisibilityDataSet1Cyclic;
	        "ProdDataInterfaceHmi".cycleTimerDataSet[2].userInterfaceVisibility := "ProdDataSimulation".ProdDataCyclic.userInterfaceVisibilityDataSet2Cyclic;
	        
	    END_IF;
	END_REGION
	
	
	REGION LimitValues
	    // Example to demonstrate and test the functionality of the limit counters
	
	    IF "ProdDataSimulation".ProdDataLimitValues.limitValuesEnable THEN
	        
	        "ProdDataInterfaceHmi".limitDataSet[1].control[1].count := "ProdDataSimulation".ProdDataLimitValues.limitVal1Count1;
	        "ProdDataInterfaceHmi".limitDataSet[1].control[1].set := "ProdDataSimulation".ProdDataLimitValues.limitVal1Set1;
	        "ProdDataSimulation".ProdDataLimitValues.limitVal1Count1PreWarn1 := "ProdDataInterfaceHmi".limitDataSet[1].control[1].prewarn;
	        "ProdDataSimulation".ProdDataLimitValues.limitVal1Count1Alarm1 := "ProdDataInterfaceHmi".limitDataSet[1].control[1].alarm;
	        "ProdDataInterfaceHmi".limitDataSet[1].control[2].count := "ProdDataSimulation".ProdDataLimitValues.limitVal1Count2;
	        "ProdDataInterfaceHmi".limitDataSet[1].control[2].set := "ProdDataSimulation".ProdDataLimitValues.limitVal1Set2;
	        "ProdDataSimulation".ProdDataLimitValues.limitVal1Count1PreWarn2 := "ProdDataInterfaceHmi".limitDataSet[1].control[2].prewarn;
	        "ProdDataSimulation".ProdDataLimitValues.limitVal1Count1Alarm2 := "ProdDataInterfaceHmi".limitDataSet[1].control[2].alarm;
	        "ProdDataInterfaceHmi".limitDataSet[1].control[3].count := "ProdDataSimulation".ProdDataLimitValues.limitVal1Count3;
	        "ProdDataInterfaceHmi".limitDataSet[1].control[3].set := "ProdDataSimulation".ProdDataLimitValues.limitVal1Set3;
	        "ProdDataSimulation".ProdDataLimitValues.limitVal1Count1PreWarn3 := "ProdDataInterfaceHmi".limitDataSet[1].control[3].prewarn;
	        "ProdDataSimulation".ProdDataLimitValues.limitVal1Count1Alarm3 := "ProdDataInterfaceHmi".limitDataSet[1].control[3].alarm;
	        
	        //Via the user interface „.userInterfaceVisibility“ [DWord] individual values can be hidden in the visualization
	        "ProdDataInterfaceHmi".limitDataSet[1].userInterfaceVisibility := "ProdDataSimulation".ProdDataLimitValues.userInterfaceVisibilityDataSet1LimitValues;
	        "ProdDataInterfaceHmi".limitDataSet[2].userInterfaceVisibility := "ProdDataSimulation".ProdDataLimitValues.userInterfaceVisibilityDataSet2LimitValues;
	    END_IF;
	END_REGION
	
	REGION ShiftCounter
	    //Example to demonstrate and test the functionality of the shift counters
	    IF "ProdDataSimulation".ProdDataShiftCounter.ShiftCounterEnable THEN
	        
	        "ProdDataInterfaceHmi".shiftCounterDataSet[1].countPartsCurrent[1] := "ProdDataSimulation".ProdDataShiftCounter.shiftCounter1Cnt1Curr;
	        "ProdDataInterfaceHmi".shiftCounterDataSet[1].countPartsCurrent[2] := "ProdDataSimulation".ProdDataShiftCounter.shiftCounter1Cnt2Curr;
	        "ProdDataInterfaceHmi".shiftCounterDataSet[1].countPartsCurrent[3] := "ProdDataSimulation".ProdDataShiftCounter.shiftCounter1Cnt3Curr;
	        "ProdDataInterfaceHmi".shiftCounterDataSet[1].resetAllExt := "ProdDataSimulation".ProdDataShiftCounter.shiftCounter1ResetAllExt;
	        
	     //Via the user interface „.userInterfaceVisibility“ [DWord] individual values can be hidden in the visualization
	        "ProdDataInterfaceHmi".shiftCounterDataSet[1].userInterfaceVisibility := "ProdDataSimulation".ProdDataShiftCounter.userInterfaceVisibilityDataSet1ShiftCounter;
	        "ProdDataInterfaceHmi".shiftCounterDataSet[2].userInterfaceVisibility := "ProdDataSimulation".ProdDataShiftCounter.userInterfaceVisibilityDataSet2ShiftCounter;
	    END_IF;
	    
	END_REGION
	
	REGION ShiftCounterOEE
	    // Example to demonstrate and test the functionality of the shift counter OEE
	    
	    IF "ProdDataSimulation".ProdDataShiftCounterOEE.ShiftCounterOEEEnable THEN
	        
	        "ProdDataInterfaceHmi".shiftCounterOeeDataSet[1].countPartsCurrent[1] := "ProdDataSimulation".ProdDataShiftCounter.shiftCounter1Cnt1Curr;
	        "ProdDataInterfaceHmi".shiftCounterOeeDataSet[1].countPartsCurrent[2] := "ProdDataSimulation".ProdDataShiftCounter.shiftCounter1Cnt2Curr;
	        "ProdDataInterfaceHmi".shiftCounterOeeDataSet[1].countPartsCurrent[3] := "ProdDataSimulation".ProdDataShiftCounter.shiftCounter1Cnt3Curr;
	        "ProdDataInterfaceHmi".shiftCounterOeeDataSet[1].countPartsCurrentOk[1] := "ProdDataSimulation".ProdDataShiftCounter.shiftCounter1Cnt1CurrOk;
	        "ProdDataInterfaceHmi".shiftCounterOeeDataSet[1].countPartsCurrentOk[2] := "ProdDataSimulation".ProdDataShiftCounter.shiftCounter1Cnt2CurrOk;
	        "ProdDataInterfaceHmi".shiftCounterOeeDataSet[1].countPartsCurrentOk[3] := "ProdDataSimulation".ProdDataShiftCounter.shiftCounter1Cnt3CurrOk;
	        
	     //Via the user interface „.userInterfaceVisibility“ [DWord] individual values can be hidden in the visualization
	        "ProdDataInterfaceHmi".shiftCounterOeeDataSet[1].userInterfaceVisibility := "ProdDataSimulation".ProdDataShiftCounterOEE.userInterfaceVisibilityDataSet1ShiftCounterOEE;
	        "ProdDataInterfaceHmi".shiftCounterOeeDataSet[2].userInterfaceVisibility := "ProdDataSimulation".ProdDataShiftCounterOEE.userInterfaceVisibilityDataSet2ShiftCounterOEE;
	    END_IF;
	END_REGION
	
	
	
END_FUNCTION

FUNCTION_BLOCK "Count"   // FB22, LAD
// stored: MemoryReserve 100, SetENOAutomatically false
   VAR
      statPulse { ExternalAccessible := 'False'; ExternalVisible := 'False'; ExternalWritable := 'False'} : Array[0..299] of Bool;
   END_VAR
   VAR_TEMP   // added for the SCL form of the ladder/FBD networks
      _w1 : Bool;
      _w2 : Bool;
      _w3 : Bool;
   END_VAR
BEGIN

REGION Network 1 (SCL): Alarms Count l Button
   // Alarm Save
   IF "Unit1.Em3.HmiInterface".topTapeCuttingCount.alarmSaveButton THEN
       "Unit1.Em3.HmiInterface".topTapeCuttingCount.ProcessValue.warningCount := "Unit1.Em3.HmiInterface".topTapeCuttingCount.SetValue.warningCount;
       "Unit1.Em3.HmiInterface".topTapeCuttingCount.ProcessValue.faultCount := "Unit1.Em3.HmiInterface".topTapeCuttingCount.SetValue.faultCount;
   END_IF;
   IF "Unit1.Em4.HmiInterface".sideTapeCuttingCount.alarmSaveButton THEN
       "Unit1.Em4.HmiInterface".sideTapeCuttingCount.ProcessValue.warningCount := "Unit1.Em4.HmiInterface".sideTapeCuttingCount.SetValue.warningCount;
       "Unit1.Em4.HmiInterface".sideTapeCuttingCount.ProcessValue.faultCount := "Unit1.Em4.HmiInterface".sideTapeCuttingCount.SetValue.faultCount;
   END_IF;
   IF "Unit1.Em9.HmiInterface".VisionNgAlarmCount.alarmSaveButton THEN
       "Unit1.Em9.HmiInterface".VisionNgAlarmCount.ProcessValue.warningCount:= "Unit1.Em9.HmiInterface".VisionNgAlarmCount.SetValue.warningCount;
       "Unit1.Em9.HmiInterface".VisionNgAlarmCount.ProcessValue.faultCount := "Unit1.Em9.HmiInterface".VisionNgAlarmCount.SetValue.faultCount;
   END_IF;


   // Count Reset
   IF "Unit1.Em3.HmiInterface".topTapeCuttingCount.countResetButton THEN
       "Unit1.Em3.HmiInterface".topTapeCuttingCount.actualCount := 0;
   END_IF;
   IF "Unit1.Em4.HmiInterface".sideTapeCuttingCount.countResetButton THEN
       "Unit1.Em4.HmiInterface".sideTapeCuttingCount.actualCount := 0;
   END_IF;
   IF "Unit1.Em9.HmiInterface".VisionNgAlarmCount.countResetButton THEN
       "Unit1.Em9.HmiInterface".VisionNgAlarmCount.actualCount := 0;
   END_IF;
END_REGION

REGION Network 2: Alarms Count l Top Tape Cutting Count Up
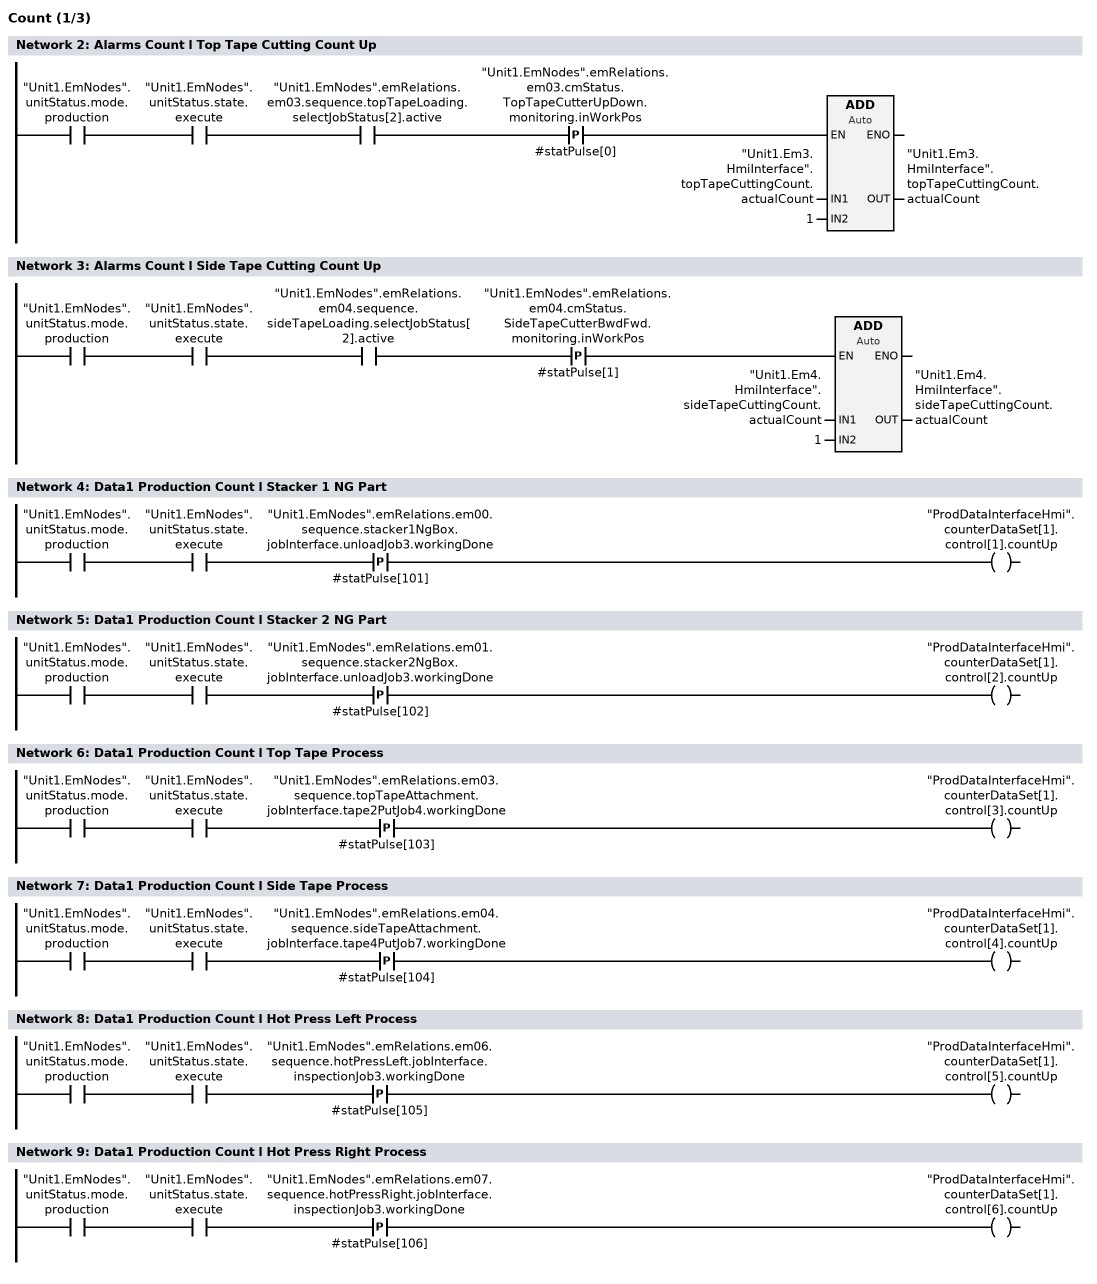
   RUNG wire#powerrail
      Contact( "Unit1.EmNodes".unitStatus.mode.production )
      Contact( "Unit1.EmNodes".unitStatus.state.execute )
      Contact( "Unit1.EmNodes".emRelations.em03.sequence.topTapeLoading.selectJobStatus[2].active )
      P_Contact(operand := "Unit1.EmNodes".emRelations.em03.cmStatus.TopTapeCutterUpDown.monitoring.inWorkPos, bit := #statPulse[0])
      Add(in1 := "Unit1.Em3.HmiInterface".topTapeCuttingCount.actualCount, in2 := 1, out => "Unit1.Em3.HmiInterface".topTapeCuttingCount.actualCount)
   END_RUNG
   // the same network as SCL:
   #_w1 := "Unit1.EmNodes".unitStatus.mode.production AND "Unit1.EmNodes".unitStatus.state.execute AND "Unit1.EmNodes".emRelations.em03.sequence.topTapeLoading.selectJobStatus[2].active AND "Unit1.EmNodes".emRelations.em03.cmStatus.TopTapeCutterUpDown.monitoring.inWorkPos AND NOT #statPulse[0];   // rising edge of "Unit1.EmNodes".emRelations.em03.cmStatus.TopTapeCutterUpDown.monitoring.inWorkPos
   #statPulse[0] := "Unit1.EmNodes".emRelations.em03.cmStatus.TopTapeCutterUpDown.monitoring.inWorkPos;
   IF #_w1 THEN
       "Unit1.Em3.HmiInterface".topTapeCuttingCount.actualCount := "Unit1.Em3.HmiInterface".topTapeCuttingCount.actualCount + 1;
   END_IF;
END_REGION

REGION Network 3: Alarms Count l Side Tape Cutting Count Up
   RUNG wire#powerrail
      Contact( "Unit1.EmNodes".unitStatus.mode.production )
      Contact( "Unit1.EmNodes".unitStatus.state.execute )
      Contact( "Unit1.EmNodes".emRelations.em04.sequence.sideTapeLoading.selectJobStatus[2].active )
      P_Contact(operand := "Unit1.EmNodes".emRelations.em04.cmStatus.SideTapeCutterBwdFwd.monitoring.inWorkPos, bit := #statPulse[1])
      Add(in1 := "Unit1.Em4.HmiInterface".sideTapeCuttingCount.actualCount, in2 := 1, out => "Unit1.Em4.HmiInterface".sideTapeCuttingCount.actualCount)
   END_RUNG
   // the same network as SCL:
   #_w1 := "Unit1.EmNodes".unitStatus.mode.production AND "Unit1.EmNodes".unitStatus.state.execute AND "Unit1.EmNodes".emRelations.em04.sequence.sideTapeLoading.selectJobStatus[2].active AND "Unit1.EmNodes".emRelations.em04.cmStatus.SideTapeCutterBwdFwd.monitoring.inWorkPos AND NOT #statPulse[1];   // rising edge of "Unit1.EmNodes".emRelations.em04.cmStatus.SideTapeCutterBwdFwd.monitoring.inWorkPos
   #statPulse[1] := "Unit1.EmNodes".emRelations.em04.cmStatus.SideTapeCutterBwdFwd.monitoring.inWorkPos;
   IF #_w1 THEN
       "Unit1.Em4.HmiInterface".sideTapeCuttingCount.actualCount := "Unit1.Em4.HmiInterface".sideTapeCuttingCount.actualCount + 1;
   END_IF;
END_REGION

REGION Network 4: Data1 Production Count l Stacker 1 NG Part
   RUNG wire#powerrail
      Contact( "Unit1.EmNodes".unitStatus.mode.production )
      Contact( "Unit1.EmNodes".unitStatus.state.execute )
      P_Contact(operand := "Unit1.EmNodes".emRelations.em00.sequence.stacker1NgBox.jobInterface.unloadJob3.workingDone, bit := #statPulse[101])
      Coil( "ProdDataInterfaceHmi".counterDataSet[1].control[1].countUp )
   END_RUNG
   // the same network as SCL:
   #_w1 := "Unit1.EmNodes".unitStatus.mode.production AND "Unit1.EmNodes".unitStatus.state.execute AND "Unit1.EmNodes".emRelations.em00.sequence.stacker1NgBox.jobInterface.unloadJob3.workingDone AND NOT #statPulse[101];   // rising edge of "Unit1.EmNodes".emRelations.em00.sequence.stacker1NgBox.jobInterface.unloadJob3.workingDone
   #statPulse[101] := "Unit1.EmNodes".emRelations.em00.sequence.stacker1NgBox.jobInterface.unloadJob3.workingDone;
   "ProdDataInterfaceHmi".counterDataSet[1].control[1].countUp := #_w1;
END_REGION

REGION Network 5: Data1 Production Count l Stacker 2 NG Part
   RUNG wire#powerrail
      Contact( "Unit1.EmNodes".unitStatus.mode.production )
      Contact( "Unit1.EmNodes".unitStatus.state.execute )
      P_Contact(operand := "Unit1.EmNodes".emRelations.em01.sequence.stacker2NgBox.jobInterface.unloadJob3.workingDone, bit := #statPulse[102])
      Coil( "ProdDataInterfaceHmi".counterDataSet[1].control[2].countUp )
   END_RUNG
   // the same network as SCL:
   #_w1 := "Unit1.EmNodes".unitStatus.mode.production AND "Unit1.EmNodes".unitStatus.state.execute AND "Unit1.EmNodes".emRelations.em01.sequence.stacker2NgBox.jobInterface.unloadJob3.workingDone AND NOT #statPulse[102];   // rising edge of "Unit1.EmNodes".emRelations.em01.sequence.stacker2NgBox.jobInterface.unloadJob3.workingDone
   #statPulse[102] := "Unit1.EmNodes".emRelations.em01.sequence.stacker2NgBox.jobInterface.unloadJob3.workingDone;
   "ProdDataInterfaceHmi".counterDataSet[1].control[2].countUp := #_w1;
END_REGION

REGION Network 6: Data1 Production Count l Top Tape Process
   RUNG wire#powerrail
      Contact( "Unit1.EmNodes".unitStatus.mode.production )
      Contact( "Unit1.EmNodes".unitStatus.state.execute )
      P_Contact(operand := "Unit1.EmNodes".emRelations.em03.sequence.topTapeAttachment.jobInterface.tape2PutJob4.workingDone, bit := #statPulse[103])
      Coil( "ProdDataInterfaceHmi".counterDataSet[1].control[3].countUp )
   END_RUNG
   // the same network as SCL:
   #_w1 := "Unit1.EmNodes".unitStatus.mode.production AND "Unit1.EmNodes".unitStatus.state.execute AND "Unit1.EmNodes".emRelations.em03.sequence.topTapeAttachment.jobInterface.tape2PutJob4.workingDone AND NOT #statPulse[103];   // rising edge of "Unit1.EmNodes".emRelations.em03.sequence.topTapeAttachment.jobInterface.tape2PutJob4.workingDone
   #statPulse[103] := "Unit1.EmNodes".emRelations.em03.sequence.topTapeAttachment.jobInterface.tape2PutJob4.workingDone;
   "ProdDataInterfaceHmi".counterDataSet[1].control[3].countUp := #_w1;
END_REGION

REGION Network 7: Data1 Production Count l Side Tape Process
   RUNG wire#powerrail
      Contact( "Unit1.EmNodes".unitStatus.mode.production )
      Contact( "Unit1.EmNodes".unitStatus.state.execute )
      P_Contact(operand := "Unit1.EmNodes".emRelations.em04.sequence.sideTapeAttachment.jobInterface.tape4PutJob7.workingDone, bit := #statPulse[104])
      Coil( "ProdDataInterfaceHmi".counterDataSet[1].control[4].countUp )
   END_RUNG
   // the same network as SCL:
   #_w1 := "Unit1.EmNodes".unitStatus.mode.production AND "Unit1.EmNodes".unitStatus.state.execute AND "Unit1.EmNodes".emRelations.em04.sequence.sideTapeAttachment.jobInterface.tape4PutJob7.workingDone AND NOT #statPulse[104];   // rising edge of "Unit1.EmNodes".emRelations.em04.sequence.sideTapeAttachment.jobInterface.tape4PutJob7.workingDone
   #statPulse[104] := "Unit1.EmNodes".emRelations.em04.sequence.sideTapeAttachment.jobInterface.tape4PutJob7.workingDone;
   "ProdDataInterfaceHmi".counterDataSet[1].control[4].countUp := #_w1;
END_REGION

REGION Network 8: Data1 Production Count l Hot Press Left Process
   RUNG wire#powerrail
      Contact( "Unit1.EmNodes".unitStatus.mode.production )
      Contact( "Unit1.EmNodes".unitStatus.state.execute )
      P_Contact(operand := "Unit1.EmNodes".emRelations.em06.sequence.hotPressLeft.jobInterface.inspectionJob3.workingDone, bit := #statPulse[105])
      Coil( "ProdDataInterfaceHmi".counterDataSet[1].control[5].countUp )
   END_RUNG
   // the same network as SCL:
   #_w1 := "Unit1.EmNodes".unitStatus.mode.production AND "Unit1.EmNodes".unitStatus.state.execute AND "Unit1.EmNodes".emRelations.em06.sequence.hotPressLeft.jobInterface.inspectionJob3.workingDone AND NOT #statPulse[105];   // rising edge of "Unit1.EmNodes".emRelations.em06.sequence.hotPressLeft.jobInterface.inspectionJob3.workingDone
   #statPulse[105] := "Unit1.EmNodes".emRelations.em06.sequence.hotPressLeft.jobInterface.inspectionJob3.workingDone;
   "ProdDataInterfaceHmi".counterDataSet[1].control[5].countUp := #_w1;
END_REGION

REGION Network 9: Data1 Production Count l Hot Press Right Process
   RUNG wire#powerrail
      Contact( "Unit1.EmNodes".unitStatus.mode.production )
      Contact( "Unit1.EmNodes".unitStatus.state.execute )
      P_Contact(operand := "Unit1.EmNodes".emRelations.em07.sequence.hotPressRight.jobInterface.inspectionJob3.workingDone, bit := #statPulse[106])
      Coil( "ProdDataInterfaceHmi".counterDataSet[1].control[6].countUp )
   END_RUNG
   // the same network as SCL:
   #_w1 := "Unit1.EmNodes".unitStatus.mode.production AND "Unit1.EmNodes".unitStatus.state.execute AND "Unit1.EmNodes".emRelations.em07.sequence.hotPressRight.jobInterface.inspectionJob3.workingDone AND NOT #statPulse[106];   // rising edge of "Unit1.EmNodes".emRelations.em07.sequence.hotPressRight.jobInterface.inspectionJob3.workingDone
   #statPulse[106] := "Unit1.EmNodes".emRelations.em07.sequence.hotPressRight.jobInterface.inspectionJob3.workingDone;
   "ProdDataInterfaceHmi".counterDataSet[1].control[6].countUp := #_w1;
END_REGION

REGION Network 10: Data1 Production Count l Hipot & Thickness Servo Press Process
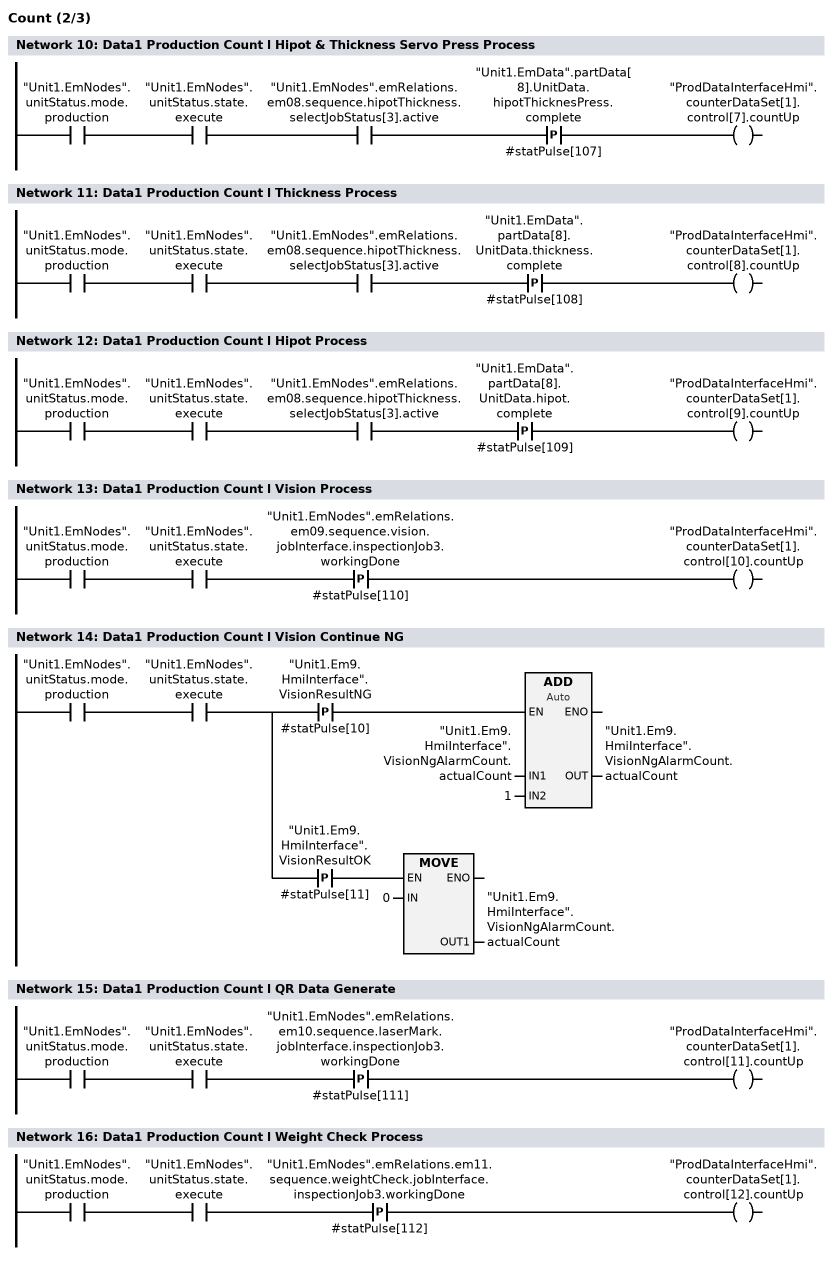
   RUNG wire#powerrail
      Contact( "Unit1.EmNodes".unitStatus.mode.production )
      Contact( "Unit1.EmNodes".unitStatus.state.execute )
      Contact( "Unit1.EmNodes".emRelations.em08.sequence.hipotThickness.selectJobStatus[3].active )
      P_Contact(operand := "Unit1.EmData".partData[8].UnitData.hipotThicknesPress.complete, bit := #statPulse[107])
      Coil( "ProdDataInterfaceHmi".counterDataSet[1].control[7].countUp )
   END_RUNG
   // the same network as SCL:
   #_w1 := "Unit1.EmNodes".unitStatus.mode.production AND "Unit1.EmNodes".unitStatus.state.execute AND "Unit1.EmNodes".emRelations.em08.sequence.hipotThickness.selectJobStatus[3].active AND "Unit1.EmData".partData[8].UnitData.hipotThicknesPress.complete AND NOT #statPulse[107];   // rising edge of "Unit1.EmData".partData[8].UnitData.hipotThicknesPress.complete
   #statPulse[107] := "Unit1.EmData".partData[8].UnitData.hipotThicknesPress.complete;
   "ProdDataInterfaceHmi".counterDataSet[1].control[7].countUp := #_w1;
END_REGION

REGION Network 11: Data1 Production Count l Thickness Process
   RUNG wire#powerrail
      Contact( "Unit1.EmNodes".unitStatus.mode.production )
      Contact( "Unit1.EmNodes".unitStatus.state.execute )
      Contact( "Unit1.EmNodes".emRelations.em08.sequence.hipotThickness.selectJobStatus[3].active )
      P_Contact(operand := "Unit1.EmData".partData[8].UnitData.thickness.complete, bit := #statPulse[108])
      Coil( "ProdDataInterfaceHmi".counterDataSet[1].control[8].countUp )
   END_RUNG
   // the same network as SCL:
   #_w1 := "Unit1.EmNodes".unitStatus.mode.production AND "Unit1.EmNodes".unitStatus.state.execute AND "Unit1.EmNodes".emRelations.em08.sequence.hipotThickness.selectJobStatus[3].active AND "Unit1.EmData".partData[8].UnitData.thickness.complete AND NOT #statPulse[108];   // rising edge of "Unit1.EmData".partData[8].UnitData.thickness.complete
   #statPulse[108] := "Unit1.EmData".partData[8].UnitData.thickness.complete;
   "ProdDataInterfaceHmi".counterDataSet[1].control[8].countUp := #_w1;
END_REGION

REGION Network 12: Data1 Production Count l Hipot Process
   RUNG wire#powerrail
      Contact( "Unit1.EmNodes".unitStatus.mode.production )
      Contact( "Unit1.EmNodes".unitStatus.state.execute )
      Contact( "Unit1.EmNodes".emRelations.em08.sequence.hipotThickness.selectJobStatus[3].active )
      P_Contact(operand := "Unit1.EmData".partData[8].UnitData.hipot.complete, bit := #statPulse[109])
      Coil( "ProdDataInterfaceHmi".counterDataSet[1].control[9].countUp )
   END_RUNG
   // the same network as SCL:
   #_w1 := "Unit1.EmNodes".unitStatus.mode.production AND "Unit1.EmNodes".unitStatus.state.execute AND "Unit1.EmNodes".emRelations.em08.sequence.hipotThickness.selectJobStatus[3].active AND "Unit1.EmData".partData[8].UnitData.hipot.complete AND NOT #statPulse[109];   // rising edge of "Unit1.EmData".partData[8].UnitData.hipot.complete
   #statPulse[109] := "Unit1.EmData".partData[8].UnitData.hipot.complete;
   "ProdDataInterfaceHmi".counterDataSet[1].control[9].countUp := #_w1;
END_REGION

REGION Network 13: Data1 Production Count l Vision Process
   RUNG wire#powerrail
      Contact( "Unit1.EmNodes".unitStatus.mode.production )
      Contact( "Unit1.EmNodes".unitStatus.state.execute )
      P_Contact(operand := "Unit1.EmNodes".emRelations.em09.sequence.vision.jobInterface.inspectionJob3.workingDone, bit := #statPulse[110])
      Coil( "ProdDataInterfaceHmi".counterDataSet[1].control[10].countUp )
   END_RUNG
   // the same network as SCL:
   #_w1 := "Unit1.EmNodes".unitStatus.mode.production AND "Unit1.EmNodes".unitStatus.state.execute AND "Unit1.EmNodes".emRelations.em09.sequence.vision.jobInterface.inspectionJob3.workingDone AND NOT #statPulse[110];   // rising edge of "Unit1.EmNodes".emRelations.em09.sequence.vision.jobInterface.inspectionJob3.workingDone
   #statPulse[110] := "Unit1.EmNodes".emRelations.em09.sequence.vision.jobInterface.inspectionJob3.workingDone;
   "ProdDataInterfaceHmi".counterDataSet[1].control[10].countUp := #_w1;
END_REGION

REGION Network 14: Data1 Production Count l Vision Continue NG
   RUNG wire#powerrail
      Contact( "Unit1.EmNodes".unitStatus.mode.production )
      Contact( "Unit1.EmNodes".unitStatus.state.execute )
      wire#w1
      P_Contact(operand := "Unit1.Em9.HmiInterface".VisionResultNG, bit := #statPulse[10])
      Add(in1 := "Unit1.Em9.HmiInterface".VisionNgAlarmCount.actualCount, in2 := 1, out => "Unit1.Em9.HmiInterface".VisionNgAlarmCount.actualCount)
   END_RUNG
   RUNG wire#w1
      P_Contact(operand := "Unit1.Em9.HmiInterface".VisionResultOK, bit := #statPulse[11])
      Move(in := 0, out1 => "Unit1.Em9.HmiInterface".VisionNgAlarmCount.actualCount)
   END_RUNG
   // the same network as SCL:
   #_w1 := "Unit1.EmNodes".unitStatus.mode.production AND "Unit1.EmNodes".unitStatus.state.execute;
   #_w2 := #_w1 AND "Unit1.Em9.HmiInterface".VisionResultNG AND NOT #statPulse[10];   // rising edge of "Unit1.Em9.HmiInterface".VisionResultNG
   #statPulse[10] := "Unit1.Em9.HmiInterface".VisionResultNG;
   IF #_w2 THEN
       "Unit1.Em9.HmiInterface".VisionNgAlarmCount.actualCount := "Unit1.Em9.HmiInterface".VisionNgAlarmCount.actualCount + 1;
   END_IF;
   #_w3 := #_w1 AND "Unit1.Em9.HmiInterface".VisionResultOK AND NOT #statPulse[11];   // rising edge of "Unit1.Em9.HmiInterface".VisionResultOK
   #statPulse[11] := "Unit1.Em9.HmiInterface".VisionResultOK;
   IF #_w3 THEN "Unit1.Em9.HmiInterface".VisionNgAlarmCount.actualCount := 0; END_IF;
END_REGION

REGION Network 15: Data1 Production Count l QR Data Generate
   RUNG wire#powerrail
      Contact( "Unit1.EmNodes".unitStatus.mode.production )
      Contact( "Unit1.EmNodes".unitStatus.state.execute )
      P_Contact(operand := "Unit1.EmNodes".emRelations.em10.sequence.laserMark.jobInterface.inspectionJob3.workingDone, bit := #statPulse[111])
      Coil( "ProdDataInterfaceHmi".counterDataSet[1].control[11].countUp )
   END_RUNG
   // the same network as SCL:
   #_w1 := "Unit1.EmNodes".unitStatus.mode.production AND "Unit1.EmNodes".unitStatus.state.execute AND "Unit1.EmNodes".emRelations.em10.sequence.laserMark.jobInterface.inspectionJob3.workingDone AND NOT #statPulse[111];   // rising edge of "Unit1.EmNodes".emRelations.em10.sequence.laserMark.jobInterface.inspectionJob3.workingDone
   #statPulse[111] := "Unit1.EmNodes".emRelations.em10.sequence.laserMark.jobInterface.inspectionJob3.workingDone;
   "ProdDataInterfaceHmi".counterDataSet[1].control[11].countUp := #_w1;
END_REGION

REGION Network 16: Data1 Production Count l Weight Check Process
   RUNG wire#powerrail
      Contact( "Unit1.EmNodes".unitStatus.mode.production )
      Contact( "Unit1.EmNodes".unitStatus.state.execute )
      P_Contact(operand := "Unit1.EmNodes".emRelations.em11.sequence.weightCheck.jobInterface.inspectionJob3.workingDone, bit := #statPulse[112])
      Coil( "ProdDataInterfaceHmi".counterDataSet[1].control[12].countUp )
   END_RUNG
   // the same network as SCL:
   #_w1 := "Unit1.EmNodes".unitStatus.mode.production AND "Unit1.EmNodes".unitStatus.state.execute AND "Unit1.EmNodes".emRelations.em11.sequence.weightCheck.jobInterface.inspectionJob3.workingDone AND NOT #statPulse[112];   // rising edge of "Unit1.EmNodes".emRelations.em11.sequence.weightCheck.jobInterface.inspectionJob3.workingDone
   #statPulse[112] := "Unit1.EmNodes".emRelations.em11.sequence.weightCheck.jobInterface.inspectionJob3.workingDone;
   "ProdDataInterfaceHmi".counterDataSet[1].control[12].countUp := #_w1;
END_REGION

REGION Network 17: Data1 Production Count l Final NG Part
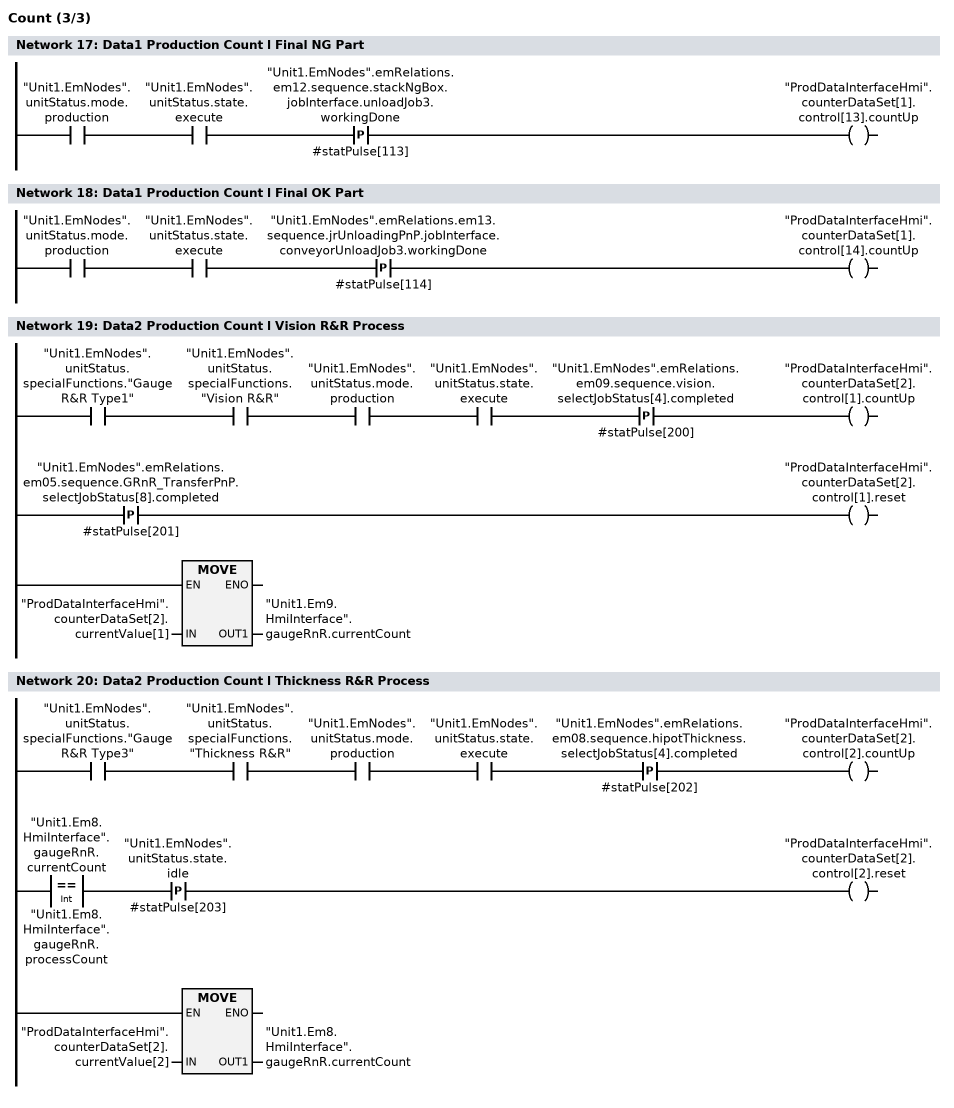
   RUNG wire#powerrail
      Contact( "Unit1.EmNodes".unitStatus.mode.production )
      Contact( "Unit1.EmNodes".unitStatus.state.execute )
      P_Contact(operand := "Unit1.EmNodes".emRelations.em12.sequence.stackNgBox.jobInterface.unloadJob3.workingDone, bit := #statPulse[113])
      Coil( "ProdDataInterfaceHmi".counterDataSet[1].control[13].countUp )
   END_RUNG
   // the same network as SCL:
   #_w1 := "Unit1.EmNodes".unitStatus.mode.production AND "Unit1.EmNodes".unitStatus.state.execute AND "Unit1.EmNodes".emRelations.em12.sequence.stackNgBox.jobInterface.unloadJob3.workingDone AND NOT #statPulse[113];   // rising edge of "Unit1.EmNodes".emRelations.em12.sequence.stackNgBox.jobInterface.unloadJob3.workingDone
   #statPulse[113] := "Unit1.EmNodes".emRelations.em12.sequence.stackNgBox.jobInterface.unloadJob3.workingDone;
   "ProdDataInterfaceHmi".counterDataSet[1].control[13].countUp := #_w1;
END_REGION

REGION Network 18: Data1 Production Count l Final OK Part
   RUNG wire#powerrail
      Contact( "Unit1.EmNodes".unitStatus.mode.production )
      Contact( "Unit1.EmNodes".unitStatus.state.execute )
      P_Contact(operand := "Unit1.EmNodes".emRelations.em13.sequence.jrUnloadingPnP.jobInterface.conveyorUnloadJob3.workingDone, bit := #statPulse[114])
      Coil( "ProdDataInterfaceHmi".counterDataSet[1].control[14].countUp )
   END_RUNG
   // the same network as SCL:
   #_w1 := "Unit1.EmNodes".unitStatus.mode.production AND "Unit1.EmNodes".unitStatus.state.execute AND "Unit1.EmNodes".emRelations.em13.sequence.jrUnloadingPnP.jobInterface.conveyorUnloadJob3.workingDone AND NOT #statPulse[114];   // rising edge of "Unit1.EmNodes".emRelations.em13.sequence.jrUnloadingPnP.jobInterface.conveyorUnloadJob3.workingDone
   #statPulse[114] := "Unit1.EmNodes".emRelations.em13.sequence.jrUnloadingPnP.jobInterface.conveyorUnloadJob3.workingDone;
   "ProdDataInterfaceHmi".counterDataSet[1].control[14].countUp := #_w1;
END_REGION

REGION Network 19: Data2 Production Count l Vision R&R Process
   RUNG wire#powerrail
      Contact( "Unit1.EmNodes".unitStatus.specialFunctions."Gauge R&R Type1" )
      Contact( "Unit1.EmNodes".unitStatus.specialFunctions."Vision R&R" )
      Contact( "Unit1.EmNodes".unitStatus.mode.production )
      Contact( "Unit1.EmNodes".unitStatus.state.execute )
      P_Contact(operand := "Unit1.EmNodes".emRelations.em09.sequence.vision.selectJobStatus[4].completed, bit := #statPulse[200])
      Coil( "ProdDataInterfaceHmi".counterDataSet[2].control[1].countUp )
   END_RUNG
   RUNG wire#powerrail
      P_Contact(operand := "Unit1.EmNodes".emRelations.em05.sequence.GRnR_TransferPnP.selectJobStatus[8].completed, bit := #statPulse[201])
      Coil( "ProdDataInterfaceHmi".counterDataSet[2].control[1].reset )
   END_RUNG
   RUNG wire#powerrail
      Move(in := "ProdDataInterfaceHmi".counterDataSet[2].currentValue[1], out1 => "Unit1.Em9.HmiInterface".gaugeRnR.currentCount)
   END_RUNG
   // the same network as SCL:
   #_w1 := "Unit1.EmNodes".unitStatus.specialFunctions."Gauge R&R Type1" AND "Unit1.EmNodes".unitStatus.specialFunctions."Vision R&R" AND "Unit1.EmNodes".unitStatus.mode.production AND "Unit1.EmNodes".unitStatus.state.execute AND "Unit1.EmNodes".emRelations.em09.sequence.vision.selectJobStatus[4].completed AND NOT #statPulse[200];   // rising edge of "Unit1.EmNodes".emRelations.em09.sequence.vision.selectJobStatus[4].completed
   #statPulse[200] := "Unit1.EmNodes".emRelations.em09.sequence.vision.selectJobStatus[4].completed;
   "ProdDataInterfaceHmi".counterDataSet[2].control[1].countUp := #_w1;
   #_w2 := "Unit1.EmNodes".emRelations.em05.sequence.GRnR_TransferPnP.selectJobStatus[8].completed AND NOT #statPulse[201];   // rising edge of "Unit1.EmNodes".emRelations.em05.sequence.GRnR_TransferPnP.selectJobStatus[8].completed
   #statPulse[201] := "Unit1.EmNodes".emRelations.em05.sequence.GRnR_TransferPnP.selectJobStatus[8].completed;
   "ProdDataInterfaceHmi".counterDataSet[2].control[1].reset := #_w2;
   "Unit1.Em9.HmiInterface".gaugeRnR.currentCount := "ProdDataInterfaceHmi".counterDataSet[2].currentValue[1];
END_REGION

REGION Network 20: Data2 Production Count l Thickness R&R Process
   RUNG wire#powerrail
      Contact( "Unit1.EmNodes".unitStatus.specialFunctions."Gauge R&R Type3" )
      Contact( "Unit1.EmNodes".unitStatus.specialFunctions."Thickness R&R" )
      Contact( "Unit1.EmNodes".unitStatus.mode.production )
      Contact( "Unit1.EmNodes".unitStatus.state.execute )
      P_Contact(operand := "Unit1.EmNodes".emRelations.em08.sequence.hipotThickness.selectJobStatus[4].completed, bit := #statPulse[202])
      Coil( "ProdDataInterfaceHmi".counterDataSet[2].control[2].countUp )
   END_RUNG
   RUNG wire#powerrail
      { S7_Templates := "SrcType := Int" } EQ_Contact(in1 := "Unit1.Em8.HmiInterface".gaugeRnR.currentCount, in2 := "Unit1.Em8.HmiInterface".gaugeRnR.processCount)
      P_Contact(operand := "Unit1.EmNodes".unitStatus.state.idle, bit := #statPulse[203])
      Coil( "ProdDataInterfaceHmi".counterDataSet[2].control[2].reset )
   END_RUNG
   RUNG wire#powerrail
      Move(in := "ProdDataInterfaceHmi".counterDataSet[2].currentValue[2], out1 => "Unit1.Em8.HmiInterface".gaugeRnR.currentCount)
   END_RUNG
   // the same network as SCL:
   #_w1 := "Unit1.EmNodes".unitStatus.specialFunctions."Gauge R&R Type3" AND "Unit1.EmNodes".unitStatus.specialFunctions."Thickness R&R" AND "Unit1.EmNodes".unitStatus.mode.production AND "Unit1.EmNodes".unitStatus.state.execute AND "Unit1.EmNodes".emRelations.em08.sequence.hipotThickness.selectJobStatus[4].completed AND NOT #statPulse[202];   // rising edge of "Unit1.EmNodes".emRelations.em08.sequence.hipotThickness.selectJobStatus[4].completed
   #statPulse[202] := "Unit1.EmNodes".emRelations.em08.sequence.hipotThickness.selectJobStatus[4].completed;
   "ProdDataInterfaceHmi".counterDataSet[2].control[2].countUp := #_w1;
   #_w2 := ("Unit1.Em8.HmiInterface".gaugeRnR.currentCount = "Unit1.Em8.HmiInterface".gaugeRnR.processCount) AND "Unit1.EmNodes".unitStatus.state.idle AND NOT #statPulse[203];   // rising edge of "Unit1.EmNodes".unitStatus.state.idle
   #statPulse[203] := "Unit1.EmNodes".unitStatus.state.idle;
   "ProdDataInterfaceHmi".counterDataSet[2].control[2].reset := #_w2;
   "Unit1.Em8.HmiInterface".gaugeRnR.currentCount := "ProdDataInterfaceHmi".counterDataSet[2].currentValue[2];
END_REGION
END_FUNCTION_BLOCK

FUNCTION_BLOCK "CompValEqOr"   // FB55, LAD
TITLE = COMP_VAL_==_OR
AUTHOR : SICAR
FAMILY : Miscellaneous
VERSION : 1.0
// Compare the values of the inputs with the value of th input _compareValue_ generating a collective OR signal from these comparisons.
// stored: IsIECCheckEnabled true, MemoryReserve 100, SetENOAutomatically true
   VAR_INPUT
      compareValue { ExternalAccessible := 'False'; ExternalVisible := 'False'; ExternalWritable := 'False'} : UInt;   // Compare value
      val1 { ExternalAccessible := 'False'; ExternalVisible := 'False'; ExternalWritable := 'False'} : UInt;   // value 1
      val2 { ExternalAccessible := 'False'; ExternalVisible := 'False'; ExternalWritable := 'False'} : UInt;   // value 2
      val3 { ExternalAccessible := 'False'; ExternalVisible := 'False'; ExternalWritable := 'False'} : UInt;   // value 3
      val4 { ExternalAccessible := 'False'; ExternalVisible := 'False'; ExternalWritable := 'False'} : UInt;   // value 4
      val5 { ExternalAccessible := 'False'; ExternalVisible := 'False'; ExternalWritable := 'False'} : UInt;   // value 5
      val6 { ExternalAccessible := 'False'; ExternalVisible := 'False'; ExternalWritable := 'False'} : UInt;   // value 6
      val7 { ExternalAccessible := 'False'; ExternalVisible := 'False'; ExternalWritable := 'False'} : UInt;   // value 7
      val8 { ExternalAccessible := 'False'; ExternalVisible := 'False'; ExternalWritable := 'False'} : UInt;   // value 8
   END_VAR
   VAR_OUTPUT
      value { ExternalAccessible := 'False'; ExternalVisible := 'False'; ExternalWritable := 'False'} : UInt;   // Result value
   END_VAR
   VAR_TEMP
      tempDummy : Bool;   // Dummy
   END_VAR
BEGIN

REGION Network 1: ChangeLog
   // SIEMENS AG / (c)Copyright 2023
   // ------------------------------------------------------------------------------
   // Title:            CompValEqOr (FB55)
   // Comment/Function: Compare the values of the inputs with the value of th input compareValue generating a collective OR signal from these comparisons.
   // Library/Family:   Automation Framework
   // Author:           Siemens Digital Industry
   // Tested with:      ---
   // Engineering:      TIA Portal V19
   // Restrictions:     -
   // Requirements:     ---
   // ------------------------------------------------------------------------------
   // Change log table:
   // Version  | Date       | Expert in charge       | Changes applied
   // ---------|------------|------------------------|------------------------------
   // 01.00.00 | 11.12.2023 | Siemens Industry Online Support
   //                         First released version
END_REGION

REGION Network 2: Description
   // The block compares the values of the inputs _in1 ... in8_ with the value of the input _compareValue_ and generates a collective OR signal from these comparisons. If at least one of the values of in1 ... in8 is equal with _compareValue_, the value of _compareValue_ is written to output “value”.  
   // Otherwise, “value” is written with the value 0.  
   // Use Case example: With this, a "summary signal" can be formed, e.g. for production data "Limit Values", with which a button can be animated (Button "ProdData", "LimitValues"). 
   // 
   // **Block call example**  
   // 
   // The call is shown as “Ladder Diagram” (LAD), without parameters.  
   // 
   // **Calling interface**  
   // 
   // The block is called in the cyclic program. In the startup projects, the block is called to generate a collective signal for the limit values of the production data. The buttons [ProdData] and [LimitValues] are animated in color, depending on the value range of the limit values.
   // 
   // **Operation mode Automatic / Manual**  
   // 
   // The block is independent of operation modes. Therefor it is not assigned to any operation mode area.
END_REGION

REGION Network 3: set VALUE = 0
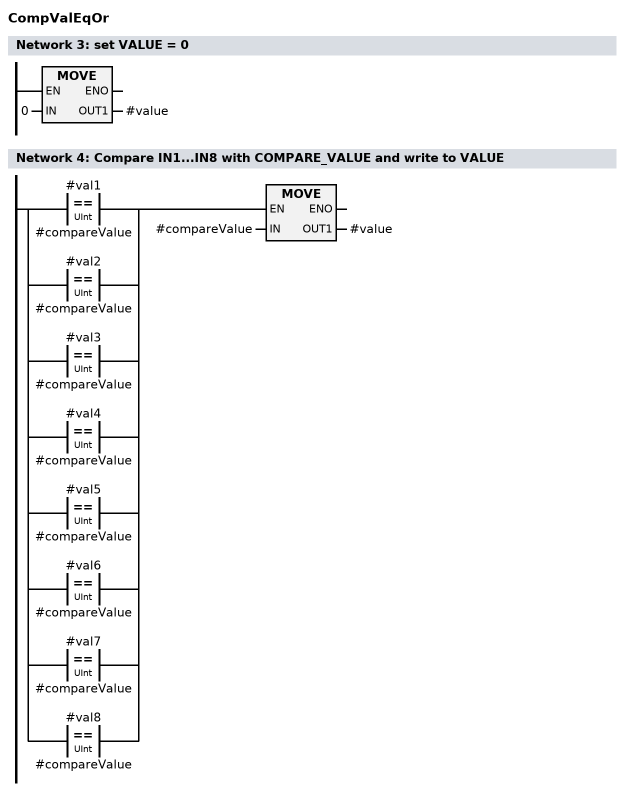
   RUNG wire#powerrail
      Move(in := 0, out1 => #value)
   END_RUNG
   // the same network as SCL:
   #value := 0;
END_REGION

REGION Network 4: Compare IN1...IN8 with COMPARE_VALUE and write to VALUE
   RUNG wire#powerrail
      { S7_Templates := "SrcType := UInt" } EQ_Contact(in1 := #val1, in2 := #compareValue)
      wire#w1
      Move(in := #compareValue, out1 => #value)
   END_RUNG
   RUNG wire#powerrail
      { S7_Templates := "SrcType := UInt" } EQ_Contact(in1 := #val2, in2 := #compareValue)
   END_RUNG wire#w1
   RUNG wire#powerrail
      { S7_Templates := "SrcType := UInt" } EQ_Contact(in1 := #val3, in2 := #compareValue)
   END_RUNG wire#w1
   RUNG wire#powerrail
      { S7_Templates := "SrcType := UInt" } EQ_Contact(in1 := #val4, in2 := #compareValue)
   END_RUNG wire#w1
   RUNG wire#powerrail
      { S7_Templates := "SrcType := UInt" } EQ_Contact(in1 := #val5, in2 := #compareValue)
   END_RUNG wire#w1
   RUNG wire#powerrail
      { S7_Templates := "SrcType := UInt" } EQ_Contact(in1 := #val6, in2 := #compareValue)
   END_RUNG wire#w1
   RUNG wire#powerrail
      { S7_Templates := "SrcType := UInt" } EQ_Contact(in1 := #val7, in2 := #compareValue)
   END_RUNG wire#w1
   RUNG wire#powerrail
      { S7_Templates := "SrcType := UInt" } EQ_Contact(in1 := #val8, in2 := #compareValue)
   END_RUNG wire#w1
   // the same network as SCL:
   IF (#val1 = #compareValue) OR (#val2 = #compareValue) OR (#val3 = #compareValue) OR (#val4 = #compareValue) OR (#val5 = #compareValue) OR (#val6 = #compareValue) OR (#val7 = #compareValue) OR (#val8 = #compareValue) THEN
       #value := #compareValue;
   END_IF;
END_REGION
END_FUNCTION_BLOCK

FUNCTION "CallEnergy" : Void   // FC5, LAD
TITLE = CallEnergy
// Call of Demo EnergyMeter and Energy Efficient M for EEMM demonstration
// stored: IsIECCheckEnabled true, SetENOAutomatically true
BEGIN

REGION Network 1: BLOCK INFO HEADER
   // SIEMENS AG / (c)Copyright 2023
   // ------------------------------------------------------------------------------
   // Title:            CallEnergy (FC5)
   // Comment/Function: Call of Demo EnergyMeter and Energy Efficient M for EEMM demonstration
   // Library/Family:   Energy
   // Author:           SICAR
   // Tested with:      ---
   // Engineering:      TIA Portal V19
   // Restrictions:     -
   // Requirements:     ---
   // ------------------------------------------------------------------------------
   // Change log table:
   // Version  | Date       | Expert in charge       | Changes applied
   // ---------|------------|------------------------|------------------------------
   // 01.00.00 | 11.12.2023 | SICAR
   //                         First released version
END_REGION

REGION Network 2: Call: Demo EnergyMeter, Energy Efficient M
   // Call for EEM demonstration
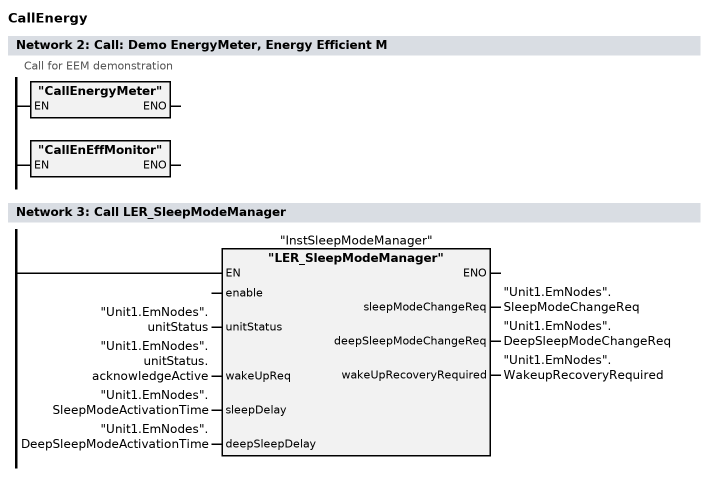
   RUNG wire#powerrail
      "CallEnergyMeter"()
   END_RUNG
   RUNG wire#powerrail
      "CallEnEffMonitor"()
   END_RUNG
   // the same network as SCL:
   "CallEnergyMeter"();
   "CallEnEffMonitor"();
END_REGION

REGION Network 3: Call LER_SleepModeManager
   RUNG wire#powerrail
      "InstSleepModeManager"(enable :=, unitStatus := "Unit1.EmNodes".unitStatus, wakeUpReq := "Unit1.EmNodes".unitStatus.acknowledgeActive, sleepDelay := "Unit1.EmNodes".SleepModeActivationTime, deepSleepDelay := "Unit1.EmNodes".DeepSleepModeActivationTime, sleepModeChangeReq => "Unit1.EmNodes".SleepModeChangeReq, deepSleepModeChangeReq => "Unit1.EmNodes".DeepSleepModeChangeReq, wakeUpRecoveryRequired => "Unit1.EmNodes".WakeupRecoveryRequired)
   END_RUNG
   // the same network as SCL:
   "InstSleepModeManager"(unitStatus := "Unit1.EmNodes".unitStatus,   // "LER_SleepModeManager"
                          wakeUpReq := "Unit1.EmNodes".unitStatus.acknowledgeActive,
                          sleepDelay := "Unit1.EmNodes".SleepModeActivationTime,
                          deepSleepDelay := "Unit1.EmNodes".DeepSleepModeActivationTime,
                          sleepModeChangeReq => "Unit1.EmNodes".SleepModeChangeReq,
                          deepSleepModeChangeReq => "Unit1.EmNodes".DeepSleepModeChangeReq,
                          wakeUpRecoveryRequired => "Unit1.EmNodes".WakeupRecoveryRequired);
END_REGION
END_FUNCTION

FUNCTION "CallEnergyMeter" : Void   // FC9, LAD
TITLE = CALL_AIEnergyMeter_FC
AUTHOR : SICAR
FAMILY : Energy
VERSION : 1.0
// This block calls the blocks for the AI-Energy-management.
// For more informations see SICAR userdefined documentation / SICAR online-help.
// stored: IsIECCheckEnabled true, SetENOAutomatically true
   VAR_TEMP
      tempCommResourceCounter : Int;   // für FB-Aufruf: E2M_1500_AIEnergyMeter_DRV
      tempBitsHmi : "typeEnMeterBits";   // für FB-Aufruf: E2M_1500_AIEnergyMeter_DRV
   END_VAR
   // Ret_Val : Ret_Val
BEGIN

REGION Network 1: ChangeLog
   // SIEMENS AG / (c)Copyright 2023
   // ------------------------------------------------------------------------------
   // Title:            CallEnergyMeter (FC9)
   // Comment/Function: This block calls the blocks for the AI-Energy-management.
   // Library/Family:   Automation Framework
   // Author:           Siemens Digital Industry
   // Tested with:      ---
   // Engineering:      TIA Portal V19
   // Restrictions:     -
   // Requirements:     ---
   // ------------------------------------------------------------------------------
   // Change log table:
   // Version  | Date       | Expert in charge       | Changes applied
   // ---------|------------|------------------------|------------------------------
   // 05.00.00 | 01.09.2023 | SICAR
   //                         First released version
END_REGION

REGION Network 2: AI_EnergyMeter 1
   // Call of E2MenergyMeterDrv FB
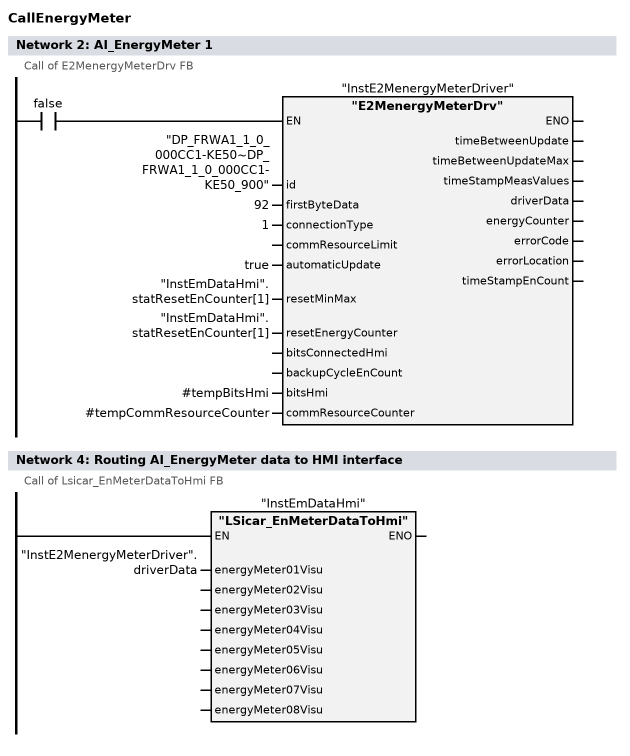
   RUNG wire#powerrail
      Contact( false )
      "InstE2MenergyMeterDriver"(id := "DP_FRWA1_1_0_000CC1-KE50~DP_FRWA1_1_0_000CC1-KE50_900", firstByteData := 92, connectionType := 1, commResourceLimit :=, automaticUpdate := true, resetMinMax := "InstEmDataHmi".statResetEnCounter[1], resetEnergyCounter := "InstEmDataHmi".statResetEnCounter[1], bitsConnectedHmi :=, backupCycleEnCount :=, bitsHmi := #tempBitsHmi, commResourceCounter := #tempCommResourceCounter, timeBetweenUpdate =>, timeBetweenUpdateMax =>, timeStampMeasValues =>, driverData =>, energyCounter =>, errorCode =>, errorLocation =>, timeStampEnCount =>)
   END_RUNG
   // the same network as SCL:
   IF false THEN
       "InstE2MenergyMeterDriver"(id := "DP_FRWA1_1_0_000CC1-KE50~DP_FRWA1_1_0_000CC1-KE50_900",   // "E2MenergyMeterDrv"
                               firstByteData := 92,
                               connectionType := 1,
                               automaticUpdate := true,
                               resetMinMax := "InstEmDataHmi".statResetEnCounter[1],
                               resetEnergyCounter := "InstEmDataHmi".statResetEnCounter[1],
                               bitsHmi := #tempBitsHmi,
                               commResourceCounter := #tempCommResourceCounter);
   END_IF;
END_REGION

REGION Network 3 (SCL): Power meter

   // Voltage L-N
   "InstE2MenergyMeterDriver".driverData.uL1 := "PAC3220InPut"."Voltage_L1-N";
   "InstE2MenergyMeterDriver".driverData.uL2 := "PAC3220InPut"."Voltage_L2-N";
   "InstE2MenergyMeterDriver".driverData.uL3 := "PAC3220InPut"."Voltage_L3-N";
   "InstE2MenergyMeterDriver".driverData.uPhNaverage :=
   ("InstE2MenergyMeterDriver".driverData.uL1 + "InstE2MenergyMeterDriver".driverData.uL2 + "InstE2MenergyMeterDriver".driverData.uL3) / 3.0;

   IF "InstE2MenergyMeterDriver".driverData.uL1 < "InstE2MenergyMeterDriver".driverData.uL1Min OR "InstE2MenergyMeterDriver".driverData.uL1Min = 0.0 THEN
       "InstE2MenergyMeterDriver".driverData.uL1Min := "InstE2MenergyMeterDriver".driverData.uL1;
   END_IF;
   IF "InstE2MenergyMeterDriver".driverData.uL1 > "InstE2MenergyMeterDriver".driverData.uL1Max OR "InstE2MenergyMeterDriver".driverData.uL1Max = 0.0 THEN
       "InstE2MenergyMeterDriver".driverData.uL1Max := "InstE2MenergyMeterDriver".driverData.uL1;
   END_IF;

   IF "InstE2MenergyMeterDriver".driverData.uL2 < "InstE2MenergyMeterDriver".driverData.uL2Min OR "InstE2MenergyMeterDriver".driverData.uL2Min = 0.0 THEN
       "InstE2MenergyMeterDriver".driverData.uL2Min := "InstE2MenergyMeterDriver".driverData.uL2;
   END_IF;
   IF "InstE2MenergyMeterDriver".driverData.uL2 > "InstE2MenergyMeterDriver".driverData.uL2Max OR "InstE2MenergyMeterDriver".driverData.uL2Max = 0.0 THEN
       "InstE2MenergyMeterDriver".driverData.uL2Max := "InstE2MenergyMeterDriver".driverData.uL2;
   END_IF;

   IF "InstE2MenergyMeterDriver".driverData.uL3 < "InstE2MenergyMeterDriver".driverData.uL3Min OR "InstE2MenergyMeterDriver".driverData.uL3Min = 0.0 THEN
       "InstE2MenergyMeterDriver".driverData.uL3Min := "InstE2MenergyMeterDriver".driverData.uL3;
   END_IF;
   IF "InstE2MenergyMeterDriver".driverData.uL3 > "InstE2MenergyMeterDriver".driverData.uL3Max OR "InstE2MenergyMeterDriver".driverData.uL3Max = 0.0 THEN
       "InstE2MenergyMeterDriver".driverData.uL3Max := "InstE2MenergyMeterDriver".driverData.uL3;
   END_IF;

   IF "InstE2MenergyMeterDriver".driverData.uPhNaverage < "InstE2MenergyMeterDriver".driverData.uPhNaverageMin OR "InstE2MenergyMeterDriver".driverData.uPhNaverageMin = 0.0 THEN
       "InstE2MenergyMeterDriver".driverData.uPhNaverageMin := "InstE2MenergyMeterDriver".driverData.uPhNaverage;
   END_IF;
   IF "InstE2MenergyMeterDriver".driverData.uPhNaverage > "InstE2MenergyMeterDriver".driverData.uPhNaverageMax OR "InstE2MenergyMeterDriver".driverData.uPhNaverageMax = 0.0 THEN
       "InstE2MenergyMeterDriver".driverData.uPhNaverageMax := "InstE2MenergyMeterDriver".driverData.uPhNaverage;
   END_IF;

   // Voltage L-L
   "InstE2MenergyMeterDriver".driverData.uL1L2 := "PAC3220InPut"."Voltage_L1-L2";
   "InstE2MenergyMeterDriver".driverData.uL2L3 := "PAC3220InPut"."Voltage_L2-L3";
   "InstE2MenergyMeterDriver".driverData.uL3L1 := "PAC3220InPut"."Voltage_L3-L1";
   "InstE2MenergyMeterDriver".driverData.uPhPhAverage :=
   ("InstE2MenergyMeterDriver".driverData.uL1L2 + "InstE2MenergyMeterDriver".driverData.uL2L3 + "InstE2MenergyMeterDriver".driverData.uL3L1) / 3.0;

   IF "InstE2MenergyMeterDriver".driverData.uL1L2 < "InstE2MenergyMeterDriver".driverData.uL1L2Min OR "InstE2MenergyMeterDriver".driverData.uL1L2Min = 0.0 THEN
       "InstE2MenergyMeterDriver".driverData.uL1L2Min := "InstE2MenergyMeterDriver".driverData.uL1L2;
   END_IF;
   IF "InstE2MenergyMeterDriver".driverData.uL1L2 > "InstE2MenergyMeterDriver".driverData.uL1L2Max OR "InstE2MenergyMeterDriver".driverData.uL1L2Max = 0.0 THEN
       "InstE2MenergyMeterDriver".driverData.uL1L2Max := "InstE2MenergyMeterDriver".driverData.uL1L2;
   END_IF;

   IF "InstE2MenergyMeterDriver".driverData.uL2L3 < "InstE2MenergyMeterDriver".driverData.uL2L3Min OR "InstE2MenergyMeterDriver".driverData.uL2L3Min = 0.0 THEN
       "InstE2MenergyMeterDriver".driverData.uL2L3Min := "InstE2MenergyMeterDriver".driverData.uL2L3;
   END_IF;
   IF "InstE2MenergyMeterDriver".driverData.uL2L3 > "InstE2MenergyMeterDriver".driverData.uL2L3Max OR "InstE2MenergyMeterDriver".driverData.uL2L3Max = 0.0 THEN
       "InstE2MenergyMeterDriver".driverData.uL2L3Max := "InstE2MenergyMeterDriver".driverData.uL2L3;
   END_IF;

   IF "InstE2MenergyMeterDriver".driverData.uL3L1 < "InstE2MenergyMeterDriver".driverData.uL3L1Min OR "InstE2MenergyMeterDriver".driverData.uL3L1Min = 0.0 THEN
       "InstE2MenergyMeterDriver".driverData.uL3L1Min := "InstE2MenergyMeterDriver".driverData.uL3L1;
   END_IF;
   IF "InstE2MenergyMeterDriver".driverData.uL3L1 > "InstE2MenergyMeterDriver".driverData.uL3L1Max OR "InstE2MenergyMeterDriver".driverData.uL3L1Max = 0.0 THEN
       "InstE2MenergyMeterDriver".driverData.uL3L1Max := "InstE2MenergyMeterDriver".driverData.uL3L1;
   END_IF;

   IF "InstE2MenergyMeterDriver".driverData.uPhPhAverage < "InstE2MenergyMeterDriver".driverData.uPhPhAverageMin OR "InstE2MenergyMeterDriver".driverData.uPhPhAverageMin = 0.0 THEN
       "InstE2MenergyMeterDriver".driverData.uPhPhAverageMin := "InstE2MenergyMeterDriver".driverData.uPhPhAverage;
   END_IF;
   IF "InstE2MenergyMeterDriver".driverData.uPhPhAverage > "InstE2MenergyMeterDriver".driverData.uPhPhAverageMax OR "InstE2MenergyMeterDriver".driverData.uPhPhAverageMax = 0.0THEN
       "InstE2MenergyMeterDriver".driverData.uPhPhAverageMax := "InstE2MenergyMeterDriver".driverData.uPhPhAverage;
   END_IF;

   // Current
   "InstE2MenergyMeterDriver".driverData.iL1 := "PAC3220InPut".Current_L1;
   "InstE2MenergyMeterDriver".driverData.iL2 := "PAC3220InPut".Current_L2;
   "InstE2MenergyMeterDriver".driverData.iL3 := "PAC3220InPut".Current_L3;
   "InstE2MenergyMeterDriver".driverData.iAverage := "PAC3220InPut"."3-phase_average_current";

   IF "InstE2MenergyMeterDriver".driverData.iL1 < "InstE2MenergyMeterDriver".driverData.iL1Min OR "InstE2MenergyMeterDriver".driverData.iL1Min = 0.0 THEN
       "InstE2MenergyMeterDriver".driverData.iL1Min := "InstE2MenergyMeterDriver".driverData.iL1;
   END_IF;
   IF "InstE2MenergyMeterDriver".driverData.iL1 > "InstE2MenergyMeterDriver".driverData.iL1Max OR "InstE2MenergyMeterDriver".driverData.iL1Max = 0.0 THEN
       "InstE2MenergyMeterDriver".driverData.iL1Max := "InstE2MenergyMeterDriver".driverData.iL1;
   END_IF;

   IF "InstE2MenergyMeterDriver".driverData.iL2 < "InstE2MenergyMeterDriver".driverData.iL2Min OR "InstE2MenergyMeterDriver".driverData.iL2Min = 0.0 THEN
       "InstE2MenergyMeterDriver".driverData.iL2Min := "InstE2MenergyMeterDriver".driverData.iL2;
   END_IF;
   IF "InstE2MenergyMeterDriver".driverData.iL2 > "InstE2MenergyMeterDriver".driverData.iL2Max OR "InstE2MenergyMeterDriver".driverData.iL2Max = 0.0 THEN
       "InstE2MenergyMeterDriver".driverData.iL2Max := "InstE2MenergyMeterDriver".driverData.iL2;
   END_IF;

   IF "InstE2MenergyMeterDriver".driverData.iL3 < "InstE2MenergyMeterDriver".driverData.iL3Min OR "InstE2MenergyMeterDriver".driverData.iL3Min = 0.0 THEN
       "InstE2MenergyMeterDriver".driverData.iL3Min := "InstE2MenergyMeterDriver".driverData.iL3;
   END_IF;
   IF "InstE2MenergyMeterDriver".driverData.iL3 > "InstE2MenergyMeterDriver".driverData.iL3Max OR "InstE2MenergyMeterDriver".driverData.iL3Max = 0.0 THEN
       "InstE2MenergyMeterDriver".driverData.iL3Max := "InstE2MenergyMeterDriver".driverData.iL3;
   END_IF;

   IF "InstE2MenergyMeterDriver".driverData.iAverage < "InstE2MenergyMeterDriver".driverData.iAverageMin OR "InstE2MenergyMeterDriver".driverData.iAverageMin = 0.0 THEN
       "InstE2MenergyMeterDriver".driverData.iAverageMin := "InstE2MenergyMeterDriver".driverData.iAverage;
   END_IF;
   IF "InstE2MenergyMeterDriver".driverData.iAverage > "InstE2MenergyMeterDriver".driverData.iAverageMax OR "InstE2MenergyMeterDriver".driverData.iAverageMax = 0.0THEN
       "InstE2MenergyMeterDriver".driverData.iAverageMax := "InstE2MenergyMeterDriver".driverData.iAverage;
   END_IF;

   // Power factor
   "InstE2MenergyMeterDriver".driverData.cosL1 := "PAC3220InPut".Power_factor_L1;
   "InstE2MenergyMeterDriver".driverData.cosL2 := "PAC3220InPut".Power_factor_L2;
   "InstE2MenergyMeterDriver".driverData.cosL3 := "PAC3220InPut".Power_factor_L3;
   "InstE2MenergyMeterDriver".driverData.cosAverage := "PAC3220InPut".Total_power_factor;

   IF "InstE2MenergyMeterDriver".driverData.cosL1 < "InstE2MenergyMeterDriver".driverData.cosL1Min OR "InstE2MenergyMeterDriver".driverData.cosL1Min = 0.0 THEN
       "InstE2MenergyMeterDriver".driverData.cosL1Min := "InstE2MenergyMeterDriver".driverData.cosL1;
   END_IF;
   IF "InstE2MenergyMeterDriver".driverData.cosL1 > "InstE2MenergyMeterDriver".driverData.cosL1Max THEN
       "InstE2MenergyMeterDriver".driverData.cosL1Max := "InstE2MenergyMeterDriver".driverData.cosL1;
   END_IF;

   IF "InstE2MenergyMeterDriver".driverData.cosL2 < "InstE2MenergyMeterDriver".driverData.cosL2Min OR "InstE2MenergyMeterDriver".driverData.cosL2Min = 0.0 THEN
       "InstE2MenergyMeterDriver".driverData.cosL2Min := "InstE2MenergyMeterDriver".driverData.cosL2;
   END_IF;
   IF "InstE2MenergyMeterDriver".driverData.cosL2 > "InstE2MenergyMeterDriver".driverData.cosL2Max OR "InstE2MenergyMeterDriver".driverData.cosL2Max = 0.0 THEN
       "InstE2MenergyMeterDriver".driverData.cosL2Max := "InstE2MenergyMeterDriver".driverData.cosL2;
   END_IF;

   IF "InstE2MenergyMeterDriver".driverData.cosL3 < "InstE2MenergyMeterDriver".driverData.cosL3Min OR "InstE2MenergyMeterDriver".driverData.cosL3Min = 0.0 THEN
       "InstE2MenergyMeterDriver".driverData.cosL3Min := "InstE2MenergyMeterDriver".driverData.cosL3;
   END_IF;
   IF "InstE2MenergyMeterDriver".driverData.cosL3 > "InstE2MenergyMeterDriver".driverData.cosL3Max OR "InstE2MenergyMeterDriver".driverData.cosL3Max = 0.0THEN
       "InstE2MenergyMeterDriver".driverData.cosL3Max := "InstE2MenergyMeterDriver".driverData.cosL3;
   END_IF;

   IF "InstE2MenergyMeterDriver".driverData.cosAverage < "InstE2MenergyMeterDriver".driverData.cosAverageMin OR "InstE2MenergyMeterDriver".driverData.cosAverageMin = 0.0 THEN
       "InstE2MenergyMeterDriver".driverData.cosAverageMin := "InstE2MenergyMeterDriver".driverData.cosAverage;
   END_IF;
   IF "InstE2MenergyMeterDriver".driverData.cosAverage > "InstE2MenergyMeterDriver".driverData.cosAverageMax OR "InstE2MenergyMeterDriver".driverData.cosAverageMax = 0.0 THEN
       "InstE2MenergyMeterDriver".driverData.cosAverageMax := "InstE2MenergyMeterDriver".driverData.cosAverage;
   END_IF;

   // Frequency
   "InstE2MenergyMeterDriver".driverData.f := "PAC3220InPut".Line_frequency;

   IF "InstE2MenergyMeterDriver".driverData.f < "InstE2MenergyMeterDriver".driverData.fMin OR "InstE2MenergyMeterDriver".driverData.fMin = 0.0 THEN
       "InstE2MenergyMeterDriver".driverData.fMin := "InstE2MenergyMeterDriver".driverData.f;
   END_IF;
   IF "InstE2MenergyMeterDriver".driverData.f > "InstE2MenergyMeterDriver".driverData.fMax OR "InstE2MenergyMeterDriver".driverData.fMax = 0.0 THEN
       "InstE2MenergyMeterDriver".driverData.fMax := "InstE2MenergyMeterDriver".driverData.f;
   END_IF;


   // Apparent power
   "InstE2MenergyMeterDriver".driverData.sL1 := "Apparent power L1";
   "InstE2MenergyMeterDriver".driverData.sL2 := "Apparent power L2";
   "InstE2MenergyMeterDriver".driverData.sL3 := "Apparent power L3";
   "InstE2MenergyMeterDriver".driverData.sTotal := "PAC3220InPut".Total_apparent_power;

   IF "InstE2MenergyMeterDriver".driverData.sL1 < "InstE2MenergyMeterDriver".driverData.sL1Min OR "InstE2MenergyMeterDriver".driverData.sL1Min = 0.0 THEN
       "InstE2MenergyMeterDriver".driverData.sL1Min := "InstE2MenergyMeterDriver".driverData.sL1;
   END_IF;
   IF "InstE2MenergyMeterDriver".driverData.sL1 > "InstE2MenergyMeterDriver".driverData.sL1Max OR "InstE2MenergyMeterDriver".driverData.sL1Max = 0.0 THEN
       "InstE2MenergyMeterDriver".driverData.sL1Max := "InstE2MenergyMeterDriver".driverData.sL1;
   END_IF;

   IF "InstE2MenergyMeterDriver".driverData.sL2 < "InstE2MenergyMeterDriver".driverData.sL2Min OR "InstE2MenergyMeterDriver".driverData.sL2Min = 0.0 THEN
       "InstE2MenergyMeterDriver".driverData.sL2Min := "InstE2MenergyMeterDriver".driverData.sL2;
   END_IF;
   IF "InstE2MenergyMeterDriver".driverData.sL2 > "InstE2MenergyMeterDriver".driverData.sL2Max OR "InstE2MenergyMeterDriver".driverData.sL2Max = 0.0 THEN
       "InstE2MenergyMeterDriver".driverData.sL2Max := "InstE2MenergyMeterDriver".driverData.sL2;
   END_IF;

   IF "InstE2MenergyMeterDriver".driverData.sL3 < "InstE2MenergyMeterDriver".driverData.sL3Min OR "InstE2MenergyMeterDriver".driverData.sL3Min = 0.0 THEN
       "InstE2MenergyMeterDriver".driverData.sL3Min := "InstE2MenergyMeterDriver".driverData.sL3;
   END_IF;
   IF "InstE2MenergyMeterDriver".driverData.sL3 > "InstE2MenergyMeterDriver".driverData.sL3Max OR "InstE2MenergyMeterDriver".driverData.sL3Max = 0.0 THEN
       "InstE2MenergyMeterDriver".driverData.sL3Max := "InstE2MenergyMeterDriver".driverData.sL3;
   END_IF;

   IF "InstE2MenergyMeterDriver".driverData.sTotal < "InstE2MenergyMeterDriver".driverData.sTotalMin OR "InstE2MenergyMeterDriver".driverData.sTotalMin = 0.0 THEN
       "InstE2MenergyMeterDriver".driverData.sTotalMin := "InstE2MenergyMeterDriver".driverData.sTotal;
   END_IF;
   IF "InstE2MenergyMeterDriver".driverData.sTotal > "InstE2MenergyMeterDriver".driverData.sTotalMax OR "InstE2MenergyMeterDriver".driverData.sTotalMax = 0.0 THEN
       "InstE2MenergyMeterDriver".driverData.sTotalMax := "InstE2MenergyMeterDriver".driverData.sTotal;
   END_IF;

   // Active power
   "InstE2MenergyMeterDriver".driverData.pL1 := "Active power L1";
   "InstE2MenergyMeterDriver".driverData.pL2 := "Active power L2";
   "InstE2MenergyMeterDriver".driverData.pL3 := "Active power L3";
   "InstE2MenergyMeterDriver".driverData.pTotal := "PAC3220InPut".Total_active_power;

   IF "InstE2MenergyMeterDriver".driverData.pL1 < "InstE2MenergyMeterDriver".driverData.pL1Min OR "InstE2MenergyMeterDriver".driverData.pL1Min = 0.0 THEN
       "InstE2MenergyMeterDriver".driverData.pL1Min := "InstE2MenergyMeterDriver".driverData.pL1;
   END_IF;
   IF "InstE2MenergyMeterDriver".driverData.pL1 > "InstE2MenergyMeterDriver".driverData.pL1Max OR "InstE2MenergyMeterDriver".driverData.pL1Max = 0.0 THEN
       "InstE2MenergyMeterDriver".driverData.pL1Max := "InstE2MenergyMeterDriver".driverData.pL1;
   END_IF;

   IF "InstE2MenergyMeterDriver".driverData.pL2 < "InstE2MenergyMeterDriver".driverData.pL2Min OR "InstE2MenergyMeterDriver".driverData.pL2Min = 0.0 THEN
       "InstE2MenergyMeterDriver".driverData.pL2Min := "InstE2MenergyMeterDriver".driverData.pL2;
   END_IF;
   IF "InstE2MenergyMeterDriver".driverData.pL2 > "InstE2MenergyMeterDriver".driverData.pL2Max OR "InstE2MenergyMeterDriver".driverData.pL2Max = 0.0 THEN
       "InstE2MenergyMeterDriver".driverData.pL2Max := "InstE2MenergyMeterDriver".driverData.pL2;
   END_IF;

   IF "InstE2MenergyMeterDriver".driverData.pL3 < "InstE2MenergyMeterDriver".driverData.pL3Min OR "InstE2MenergyMeterDriver".driverData.pL3Min = 0.0 THEN
       "InstE2MenergyMeterDriver".driverData.pL3Min := "InstE2MenergyMeterDriver".driverData.pL3;
   END_IF;
   IF "InstE2MenergyMeterDriver".driverData.pL3 > "InstE2MenergyMeterDriver".driverData.pL3Max OR "InstE2MenergyMeterDriver".driverData.pL3Max = 0.0 THEN
       "InstE2MenergyMeterDriver".driverData.pL3Max := "InstE2MenergyMeterDriver".driverData.pL3;
   END_IF;

   IF "InstE2MenergyMeterDriver".driverData.pTotal < "InstE2MenergyMeterDriver".driverData.pTotalMin OR "InstE2MenergyMeterDriver".driverData.pTotalMin = 0.0 THEN
       "InstE2MenergyMeterDriver".driverData.pTotalMin := "InstE2MenergyMeterDriver".driverData.pTotal;
   END_IF;
   IF "InstE2MenergyMeterDriver".driverData.pTotal > "InstE2MenergyMeterDriver".driverData.pTotalMax OR "InstE2MenergyMeterDriver".driverData.pTotalMax = 0.0 THEN
       "InstE2MenergyMeterDriver".driverData.pTotalMax := "InstE2MenergyMeterDriver".driverData.pTotal;
   END_IF;

   // Reactive power
   "InstE2MenergyMeterDriver".driverData.qL1 := "Reactive power L1";
   "InstE2MenergyMeterDriver".driverData.qL2 := "Reactive power L2";
   "InstE2MenergyMeterDriver".driverData.qL3 := "Reactive power L3";
   "InstE2MenergyMeterDriver".driverData.qTotal := "PAC3220InPut"."Total_reactive_power_(VARn)";

   IF "InstE2MenergyMeterDriver".driverData.qL1 < "InstE2MenergyMeterDriver".driverData.qL1Min OR "InstE2MenergyMeterDriver".driverData.qL1Min = 0.0 THEN
       "InstE2MenergyMeterDriver".driverData.qL1Min := "InstE2MenergyMeterDriver".driverData.qL1;
   END_IF;
   IF "InstE2MenergyMeterDriver".driverData.qL1 > "InstE2MenergyMeterDriver".driverData.qL1Max OR "InstE2MenergyMeterDriver".driverData.qL1Max = 0.0 THEN
       "InstE2MenergyMeterDriver".driverData.qL1Max := "InstE2MenergyMeterDriver".driverData.qL1;
   END_IF;

   IF "InstE2MenergyMeterDriver".driverData.qL2 < "InstE2MenergyMeterDriver".driverData.qL2Min OR "InstE2MenergyMeterDriver".driverData.qL2Min = 0.0 THEN
       "InstE2MenergyMeterDriver".driverData.qL2Min := "InstE2MenergyMeterDriver".driverData.qL2;
   END_IF;
   IF "InstE2MenergyMeterDriver".driverData.qL2 > "InstE2MenergyMeterDriver".driverData.qL2Max OR "InstE2MenergyMeterDriver".driverData.qL2Max = 0.0 THEN
       "InstE2MenergyMeterDriver".driverData.qL2Max := "InstE2MenergyMeterDriver".driverData.qL2;
   END_IF;

   IF "InstE2MenergyMeterDriver".driverData.qL3 < "InstE2MenergyMeterDriver".driverData.qL3Min OR "InstE2MenergyMeterDriver".driverData.qL3Min = 0.0 THEN
       "InstE2MenergyMeterDriver".driverData.qL3Min := "InstE2MenergyMeterDriver".driverData.qL3;
   END_IF;
   IF "InstE2MenergyMeterDriver".driverData.qL3 > "InstE2MenergyMeterDriver".driverData.qL3Max OR "InstE2MenergyMeterDriver".driverData.qL3Max = 0.0 THEN
       "InstE2MenergyMeterDriver".driverData.qL3Max := "InstE2MenergyMeterDriver".driverData.qL3;
   END_IF;

   IF "InstE2MenergyMeterDriver".driverData.qTotal < "InstE2MenergyMeterDriver".driverData.qTotalMin OR "InstE2MenergyMeterDriver".driverData.qTotalMin = 0.0 THEN
       "InstE2MenergyMeterDriver".driverData.qTotalMin := "InstE2MenergyMeterDriver".driverData.qTotal;
   END_IF;
   IF "InstE2MenergyMeterDriver".driverData.qTotal > "InstE2MenergyMeterDriver".driverData.qTotalMax OR "InstE2MenergyMeterDriver".driverData.qTotalMax = 0.0 THEN
       "InstE2MenergyMeterDriver".driverData.qTotalMax := "InstE2MenergyMeterDriver".driverData.qTotal;
   END_IF;

   // Energy Tarif
   "InstE2MenergyMeterDriver".driverData.eActiveRate1Import := "Active energy import tariff 1(F)";
   "InstE2MenergyMeterDriver".driverData.eReactiveRate1Import := "Reactive energy import tariff 1 (F)";
   "InstE2MenergyMeterDriver".driverData.eApparentRate1Import := "Apparent energy tariff 1 (F)";
   "InstE2MenergyMeterDriver".driverData.eActiveRate1Export := "Active energy export tariff 1(F)";
   "InstE2MenergyMeterDriver".driverData.eReactiveRate1Export := "Reactive energy export tariff 1 (F)";






   // Reset 
   IF "InstEmDataHmi".statResetMinMaxAll  THEN

       // 모든 Min/Max 초기화 (Actual 값으로)
       "InstE2MenergyMeterDriver".driverData.uL1Min := 0.0;
       "InstE2MenergyMeterDriver".driverData.uL1Max := 0.0;
       "InstE2MenergyMeterDriver".driverData.uL2Min := 0.0;
       "InstE2MenergyMeterDriver".driverData.uL2Max := 0.0;
       "InstE2MenergyMeterDriver".driverData.uL3Min := 0.0;
       "InstE2MenergyMeterDriver".driverData.uL3Max := 0.0;

       "InstE2MenergyMeterDriver".driverData.uL1L2Min := 0.0;
       "InstE2MenergyMeterDriver".driverData.uL1L2Max := 0.0;
       "InstE2MenergyMeterDriver".driverData.uL2L3Min := 0.0;
       "InstE2MenergyMeterDriver".driverData.uL2L3Max := 0.0;
       "InstE2MenergyMeterDriver".driverData.uL3L1Min := 0.0;
       "InstE2MenergyMeterDriver".driverData.uL3L1Max := 0.0;

       "InstE2MenergyMeterDriver".driverData.uPhNaverageMin := 0.0;
       "InstE2MenergyMeterDriver".driverData.uPhNaverageMax := 0.0;

       "InstE2MenergyMeterDriver".driverData.uPhPhAverageMin := 0.0;
       "InstE2MenergyMeterDriver".driverData.uPhPhAverageMax := 0.0;

       "InstE2MenergyMeterDriver".driverData.iL1Min := 0.0;
       "InstE2MenergyMeterDriver".driverData.iL1Max := 0.0;
       "InstE2MenergyMeterDriver".driverData.iL2Min := 0.0;
       "InstE2MenergyMeterDriver".driverData.iL2Max := 0.0;
       "InstE2MenergyMeterDriver".driverData.iL3Min := 0.0;
       "InstE2MenergyMeterDriver".driverData.iL3Max := 0.0;

       "InstE2MenergyMeterDriver".driverData.iAverageMin := 0.0;
       "InstE2MenergyMeterDriver".driverData.iAverageMax := 0.0;

       "InstE2MenergyMeterDriver".driverData.cosL1Min := 0.0;
       "InstE2MenergyMeterDriver".driverData.cosL1Max := 0.0;
       "InstE2MenergyMeterDriver".driverData.cosL2Min := 0.0;
       "InstE2MenergyMeterDriver".driverData.cosL2Max := 0.0;
       "InstE2MenergyMeterDriver".driverData.cosL3Min := 0.0;
       "InstE2MenergyMeterDriver".driverData.cosL3Max := 0.0;

       "InstE2MenergyMeterDriver".driverData.cosAverageMin := 0.0;
       "InstE2MenergyMeterDriver".driverData.cosAverageMax := 0.0;

       "InstE2MenergyMeterDriver".driverData.fMin := 0.0;
       "InstE2MenergyMeterDriver".driverData.fMax := 0.0;

       "InstE2MenergyMeterDriver".driverData.pTotalMin := 0.0;
       "InstE2MenergyMeterDriver".driverData.pTotalMax := 0.0;
       "InstE2MenergyMeterDriver".driverData.qTotalMin := 0.0;
       "InstE2MenergyMeterDriver".driverData.qTotalMax := 0.0;
       "InstE2MenergyMeterDriver".driverData.sTotalMin := 0.0;
       "InstE2MenergyMeterDriver".driverData.sTotalMax := 0.0;

       "InstE2MenergyMeterDriver".driverData.sL1Min := 0.0;
       "InstE2MenergyMeterDriver".driverData.sL1Max := 0.0;
       "InstE2MenergyMeterDriver".driverData.sL2Min := 0.0;
       "InstE2MenergyMeterDriver".driverData.sL2Max := 0.0;
       "InstE2MenergyMeterDriver".driverData.sL3Min := 0.0;
       "InstE2MenergyMeterDriver".driverData.sL3Max := 0.0;

